KUKA KRL program: MyProgram_009().src

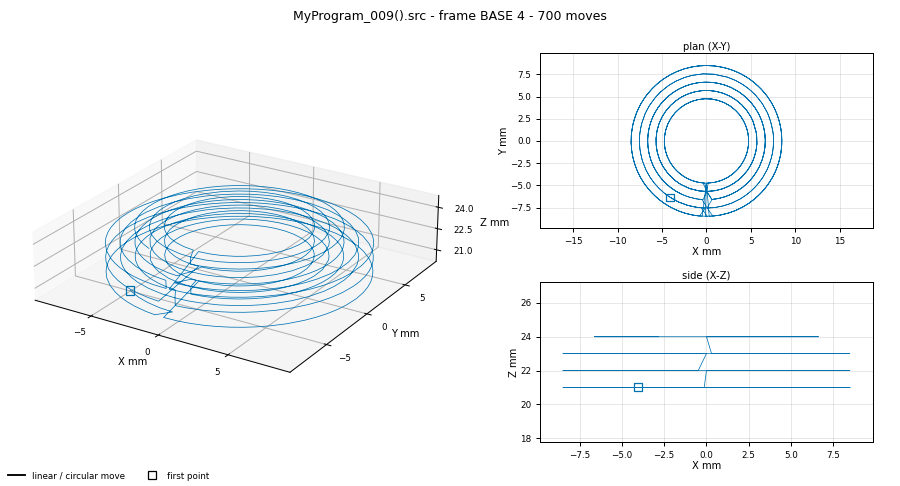
[picture p0: tool path of MyProgram_009().src in frame BASE 4, 700 of 700 moves have a stored position in this frame; points joined in program order, loops and branches not executed]
&ACCESS RVP
&REL 1
&PARAM TEMPLATE = C:\KRC\Roboter\Template\vorgabe
&PARAM EDITMASK = *
DEF MyProgram_009()
; ---- Setting reference (Base) ----
$BASE = BASE_DATA[4]

; --------------------------
; ---- Setting tool (TCP) ----
$TOOL = TOOL_DATA[3]
; --------------------------

$VEL.CP = VEL_APROX_PRINT
Startdeposition()
$VEL.CP = VEL_PRINT
LIN {X -4.0683,Y -6.363,Z 21,A -3.1712,B 0,C 0,E1 0.1598,E2 90.0712} C_DIS
LIN {X -3.0354,Y -6.9206,Z 21,A -3.1569,B 0,C 0,E1 0.1598,E2 90.0712} C_DIS
LIN {X -2.1485,Y -7.2456,Z 21,A -3.1382,B 0,C 0,E1 0.1598,E2 90.0713} C_DIS
LIN {X -1.0791,Y -7.4803,Z 21,A -3.109,B 0,C 0,E1 0.1598,E2 90.0713} C_DIS
LIN {X -0.0999,Y -7.555,Z 21,A -3.0763,B 0,C 0,E1 0.1598,E2 90.0715} C_DIS
Enddeposition()
LIN {X -0.0999,Y -7.555,Z 21,A -3.0763,B 0,C 0,E1 0.1598,E2 90.0715} C_DIS
Startdeposition()
$VEL.CP = VEL_PRINT
LIN {X -0.7948,Y -8.4503,Z 21,A -3.1394,B 0,C 0,E1 0.1598,E2 90.0708} C_DIS
LIN {X -1.524,Y -8.3542,Z 21,A -3.1626,B 0,C 0,E1 0.1598,E2 90.0713} C_DIS
LIN {X -2.5177,Y -8.1076,Z 21,A -3.1885,B 0,C 0,E1 0.1598,E2 90.0713} C_DIS
LIN {X -3.2872,Y -7.8268,Z 21,A -3.2048,B 0,C 0,E1 0.1598,E2 90.0713} C_DIS
LIN {X -4.0259,Y -7.4729,Z 21,A -3.2169,B 0,C 0,E1 0.1598,E2 90.0713} C_DIS
LIN {X -4.7269,Y -7.0495,Z 21,A -3.2247,B 0,C 0,E1 0.1598,E2 90.0712} C_DIS
LIN {X -5.5428,Y -6.4311,Z 21,A -3.2283,B 0,C 0,E1 0.1598,E2 90.071} C_DIS
LIN {X -6.3573,Y -5.629,Z 21,A -3.2241,B 0,C 0,E1 0.1598,E2 90.071} C_DIS
LIN {X -6.9724,Y -4.8392,Z 21,A -3.2134,B 0,C 0,E1 0.1598,E2 90.071} C_DIS
LIN {X -7.3967,Y -4.1598,Z 21,A -3.2003,B 0,C 0,E1 0.1598,E2 90.071} C_DIS
LIN {X -7.7565,Y -3.4443,Z 21,A -3.1833,B 0,C 0,E1 0.1598,E2 90.071} C_DIS
LIN {X -8.0474,Y -2.698,Z 21,A -3.1625,B 0,C 0,E1 0.1598,E2 90.071} C_DIS
LIN {X -8.2655,Y -1.9273,Z 21,A -3.138,B 0,C 0,E1 0.1598,E2 90.071} C_DIS
LIN {X -8.4101,Y -1.1396,Z 21,A -3.1101,B 0,C 0,E1 0.1598,E2 90.0711} C_DIS
LIN {X -8.4806,Y -0.3418,Z 21,A -3.079,B 0,C 0,E1 0.1598,E2 90.0711} C_DIS
LIN {X -8.4653,Y 0.6591,Z 21,A -3.036,B 0,C 0,E1 0.1598,E2 90.0709} C_DIS
LIN {X -8.2847,Y 1.8443,Z 21,A -2.9793,B 0,C 0,E1 0.1598,E2 90.0709} C_DIS
LIN {X -8.0734,Y 2.6138,Z 21,A -2.9395,B 0,C 0,E1 0.1598,E2 90.0713} C_DIS
LIN {X -7.7917,Y 3.3604,Z 21,A -2.8977,B 0,C 0,E1 0.1598,E2 90.0714} C_DIS
LIN {X -7.4414,Y 4.0773,Z 21,A -2.8546,B 0,C 0,E1 0.1598,E2 90.0715} C_DIS
LIN {X -7.0277,Y 4.7596,Z 21,A -2.8106,B 0,C 0,E1 0.1598,E2 90.0715} C_DIS
LIN {X -6.549,Y 5.3982,Z 21,A -2.7661,B 0,C 0,E1 0.1598,E2 90.0717} C_DIS
LIN {X -5.7701,Y 6.2287,Z 21,A -2.7022,B 0,C 0,E1 0.1598,E2 90.0717} C_DIS
LIN {X -4.9804,Y 6.8782,Z 21,A -2.6458,B 0,C 0,E1 0.1598,E2 90.0718} C_DIS
LIN {X -4.0916,Y 7.4385,Z 21,A -2.5895,B 0,C 0,E1 0.1598,E2 90.072} C_DIS
LIN {X -3.3359,Y 7.8065,Z 21,A -2.5461,B 0,C 0,E1 0.1598,E2 90.0721} C_DIS
LIN {X -2.5475,Y 8.0981,Z 21,A -2.5047,B 0,C 0,E1 0.1598,E2 90.0721} C_DIS
LIN {X -1.7342,Y 8.3101,Z 21,A -2.4658,B 0,C 0,E1 0.1598,E2 90.0723} C_DIS
LIN {X -0.9038,Y 8.44,Z 21,A -2.4296,B 0,C 0,E1 0.1598,E2 90.0723} C_DIS
LIN {X -0.0646,Y 8.4866,Z 21,A -2.3967,B 0,C 0,E1 0.1598,E2 90.0723} C_DIS
LIN {X 0.7752,Y 8.4513,Z 21,A -2.3671,B 0,C 0,E1 0.1598,E2 90.0724} C_DIS
LIN {X 1.6073,Y 8.3337,Z 21,A -2.3414,B 0,C 0,E1 0.1598,E2 90.0724} C_DIS
LIN {X 2.4237,Y 8.1342,Z 21,A -2.3196,B 0,C 0,E1 0.1598,E2 90.0724} C_DIS
LIN {X 3.2162,Y 7.8546,Z 21,A -2.3022,B 0,C 0,E1 0.1598,E2 90.0724} C_DIS
LIN {X 3.9771,Y 7.498,Z 21,A -2.2892,B 0,C 0,E1 0.1598,E2 90.0724} C_DIS
LIN {X 4.6991,Y 7.0679,Z 21,A -2.2807,B 0,C 0,E1 0.1598,E2 90.0724} C_DIS
LIN {X 5.3751,Y 6.5684,Z 21,A -2.2769,B 0,C 0,E1 0.1598,E2 90.0724} C_DIS
LIN {X 6.2322,Y 5.7664,Z 21,A -2.2791,B 0,C 0,E1 0.1598,E2 90.0722} C_DIS
LIN {X 6.8932,Y 4.9521,Z 21,A -2.2893,B 0,C 0,E1 0.1598,E2 90.0722} C_DIS
LIN {X 7.3483,Y 4.2471,Z 21,A -2.3025,B 0,C 0,E1 0.1598,E2 90.0722} C_DIS
LIN {X 7.7317,Y 3.5007,Z 21,A -2.3201,B 0,C 0,E1 0.1598,E2 90.0722} C_DIS
LIN {X 8.0395,Y 2.7201,Z 21,A -2.3419,B 0,C 0,E1 0.1598,E2 90.0721} C_DIS
LIN {X 8.2688,Y 1.913,Z 21,A -2.3677,B 0,C 0,E1 0.1598,E2 90.0721} C_DIS
LIN {X 8.4177,Y 1.0873,Z 21,A -2.3974,B 0,C 0,E1 0.1598,E2 90.072} C_DIS
LIN {X 8.4918,Y 0.0412,Z 21,A -2.4388,B 0,C 0,E1 0.1598,E2 90.0716} C_DIS
LIN {X 8.4127,Y -1.1163,Z 21,A -2.4909,B 0,C 0,E1 0.1598,E2 90.0715} C_DIS
LIN {X 8.2597,Y -1.9478,Z 21,A -2.5323,B 0,C 0,E1 0.1598,E2 90.0718} C_DIS
LIN {X 8.0253,Y -2.7601,Z 21,A -2.5755,B 0,C 0,E1 0.1598,E2 90.0718} C_DIS
LIN {X 7.7111,Y -3.5449,Z 21,A -2.6205,B 0,C 0,E1 0.1598,E2 90.0718} C_DIS
LIN {X 7.3199,Y -4.2944,Z 21,A -2.6668,B 0,C 0,E1 0.1598,E2 90.0718} C_DIS
LIN {X 6.6511,Y -5.2781,Z 21,A -2.733,B 0,C 0,E1 0.1598,E2 90.0715} C_DIS
LIN {X 5.9658,Y -6.0366,Z 21,A -2.7906,B 0,C 0,E1 0.1598,E2 90.0715} C_DIS
LIN {X 5.3564,Y -6.5819,Z 21,A -2.8363,B 0,C 0,E1 0.1598,E2 90.0716} C_DIS
LIN {X 4.6979,Y -7.0665,Z 21,A -2.8811,B 0,C 0,E1 0.1598,E2 90.0716} C_DIS
LIN {X 3.9958,Y -7.4856,Z 21,A -2.9247,B 0,C 0,E1 0.1598,E2 90.0716} C_DIS
LIN {X 3.2567,Y -7.8353,Z 21,A -2.9667,B 0,C 0,E1 0.1598,E2 90.0716} C_DIS
LIN {X 2.4875,Y -8.1124,Z 21,A -3.0067,B 0,C 0,E1 0.1598,E2 90.0716} C_DIS
LIN {X 1.6953,Y -8.3144,Z 21,A -3.0443,B 0,C 0,E1 0.1598,E2 90.0716} C_DIS
LIN {X 0.8873,Y -8.4397,Z 21,A -3.0793,B 0,C 0,E1 0.1598,E2 90.0715} C_DIS
LIN {X -0.1334,Y -8.4872,Z 21,A -3.1187,B 0,C 0,E1 0.1598,E2 90.0715} C_DIS
Enddeposition()
LIN {X 0.0005,Y -4.7572,Z 22,A -2.9405,B 0,C 0,E1 0.1598,E2 90.0604} C_DIS
Startdeposition()
$VEL.CP = VEL_PRINT
LIN {X 0.0005,Y -4.7572,Z 22,A -2.9462,B 0,C 0,E1 0.1598,E2 90.0661} C_DIS
LIN {X 0.9506,Y -4.6543,Z 22,A -2.9118,B 0,C 0,E1 0.1598,E2 90.071} C_DIS
LIN {X 1.6849,Y -4.4415,Z 22,A -2.8764,B 0,C 0,E1 0.1598,E2 90.0717} C_DIS
LIN {X 2.3764,Y -4.1152,Z 22,A -2.8372,B 0,C 0,E1 0.1598,E2 90.0717} C_DIS
LIN {X 3.0053,Y -3.68,Z 22,A -2.7955,B 0,C 0,E1 0.1598,E2 90.0717} C_DIS
LIN {X 3.5547,Y -3.1485,Z 22,A -2.7527,B 0,C 0,E1 0.1598,E2 90.0717} C_DIS
LIN {X 4.0149,Y -2.5382,Z 22,A -2.7099,B 0,C 0,E1 0.1598,E2 90.0717} C_DIS
LIN {X 4.37,Y -1.8612,Z 22,A -2.668,B 0,C 0,E1 0.1598,E2 90.0717} C_DIS
LIN {X 4.6111,Y -1.1359,Z 22,A -2.6283,B 0,C 0,E1 0.1598,E2 90.0717} C_DIS
LIN {X 4.734,Y -0.3815,Z 22,A -2.5917,B 0,C 0,E1 0.1598,E2 90.0718} C_DIS
LIN {X 4.7337,Y 0.3827,Z 22,A -2.5592,B 0,C 0,E1 0.1598,E2 90.0718} C_DIS
LIN {X 4.6108,Y 1.137,Z 22,A -2.5317,B 0,C 0,E1 0.1598,E2 90.0718} C_DIS
LIN {X 4.3693,Y 1.8622,Z 22,A -2.5099,B 0,C 0,E1 0.1598,E2 90.0719} C_DIS
LIN {X 4.0142,Y 2.5391,Z 22,A -2.4942,B 0,C 0,E1 0.1598,E2 90.0719} C_DIS
LIN {X 3.679,Y 3.0044,Z 22,A -2.487,B 0,C 0,E1 0.1598,E2 90.0721} C_DIS
LIN {X 3.1484,Y 3.5548,Z 22,A -2.4831,B 0,C 0,E1 0.1598,E2 90.0721} C_DIS
LIN {X 2.6975,Y 3.9089,Z 22,A -2.4848,B 0,C 0,E1 0.1598,E2 90.0721} C_DIS
LIN {X 2.0353,Y 4.2907,Z 22,A -2.4931,B 0,C 0,E1 0.1598,E2 90.0721} C_DIS
LIN {X 1.3208,Y 4.5621,Z 22,A -2.508,B 0,C 0,E1 0.1598,E2 90.0721} C_DIS
LIN {X 0.5721,Y 4.7168,Z 22,A -2.529,B 0,C 0,E1 0.1598,E2 90.0721} C_DIS
LIN {X -0.1919,Y 4.7486,Z 22,A -2.5559,B 0,C 0,E1 0.1598,E2 90.0721} C_DIS
LIN {X -0.9507,Y 4.6542,Z 22,A -2.5878,B 0,C 0,E1 0.1598,E2 90.0721} C_DIS
LIN {X -1.6845,Y 4.4401,Z 22,A -2.6239,B 0,C 0,E1 0.1598,E2 90.0721} C_DIS
LIN {X -2.3747,Y 4.112,Z 22,A -2.6632,B 0,C 0,E1 0.1598,E2 90.072} C_DIS
LIN {X -3.0046,Y 3.6789,Z 22,A -2.7047,B 0,C 0,E1 0.1598,E2 90.0719} C_DIS
LIN {X -3.5548,Y 3.1485,Z 22,A -2.7473,B 0,C 0,E1 0.1598,E2 90.0718} C_DIS
LIN {X -4.0153,Y 2.5384,Z 22,A -2.79,B 0,C 0,E1 0.1598,E2 90.0717} C_DIS
LIN {X -4.3701,Y 1.8612,Z 22,A -2.8316,B 0,C 0,E1 0.1598,E2 90.0716} C_DIS
LIN {X -4.6111,Y 1.1358,Z 22,A -2.8711,B 0,C 0,E1 0.1598,E2 90.0715} C_DIS
LIN {X -4.734,Y 0.3815,Z 22,A -2.9074,B 0,C 0,E1 0.1598,E2 90.0715} C_DIS
LIN {X -4.7346,Y -0.3828,Z 22,A -2.9397,B 0,C 0,E1 0.1598,E2 90.0713} C_DIS
LIN {X -4.611,Y -1.137,Z 22,A -2.967,B 0,C 0,E1 0.1598,E2 90.0713} C_DIS
LIN {X -4.3699,Y -1.8624,Z 22,A -2.9888,B 0,C 0,E1 0.1598,E2 90.0713} C_DIS
LIN {X -4.0147,Y -2.5393,Z 22,A -3.0044,B 0,C 0,E1 0.1598,E2 90.0713} C_DIS
LIN {X -3.5544,Y -3.1496,Z 22,A -3.0134,B 0,C 0,E1 0.1598,E2 90.0713} C_DIS
LIN {X -3.0038,Y -3.6798,Z 22,A -3.0156,B 0,C 0,E1 0.1598,E2 90.0713} C_DIS
LIN {X -2.3737,Y -4.1126,Z 22,A -3.0109,B 0,C 0,E1 0.1598,E2 90.0715} C_DIS
LIN {X -1.6836,Y -4.4408,Z 22,A -2.9995,B 0,C 0,E1 0.1598,E2 90.0715} C_DIS
LIN {X -0.9496,Y -4.6545,Z 22,A -2.9816,B 0,C 0,E1 0.1598,E2 90.0715} C_DIS
LIN {X -0.1908,Y -4.7488,Z 22,A -2.9578,B 0,C 0,E1 0.1598,E2 90.0716} C_DIS
LIN {X -0.1908,Y -4.7488,Z 22,A -2.9578,B 0,C 0,E1 0.1598,E2 90.0716} C_DIS
Enddeposition()
LIN {X 0.0239,Y -5.6874,Z 22,A -2.9887,B 0,C 0,E1 0.1598,E2 90.0704} C_DIS
Startdeposition()
$VEL.CP = VEL_PRINT
LIN {X -0.9077,Y -5.6101,Z 22,A -3.0207,B 0,C 0,E1 0.1598,E2 90.0715} C_DIS
LIN {X -1.8174,Y -5.3928,Z 22,A -3.0449,B 0,C 0,E1 0.1598,E2 90.0715} C_DIS
LIN {X -2.8689,Y -4.9093,Z 22,A -3.0629,B 0,C 0,E1 0.1598,E2 90.0714} C_DIS
LIN {X -3.4854,Y -4.493,Z 22,A -3.0679,B 0,C 0,E1 0.1598,E2 90.0714} C_DIS
LIN {X -4.2717,Y -3.7584,Z 22,A -3.0655,B 0,C 0,E1 0.1598,E2 90.0712} C_DIS
LIN {X -4.9659,Y -2.7683,Z 22,A -3.0489,B 0,C 0,E1 0.1598,E2 90.071} C_DIS
LIN {X -5.3072,Y -2.0335,Z 22,A -3.0306,B 0,C 0,E1 0.1598,E2 90.0712} C_DIS
LIN {X -5.5422,Y -1.2582,Z 22,A -3.0065,B 0,C 0,E1 0.1598,E2 90.0712} C_DIS
LIN {X -5.6647,Y -0.4576,Z 22,A -2.9772,B 0,C 0,E1 0.1598,E2 90.0712} C_DIS
LIN {X -5.671,Y 0.3523,Z 22,A -2.9432,B 0,C 0,E1 0.1598,E2 90.0713} C_DIS
LIN {X -5.5643,Y 1.1551,Z 22,A -2.9054,B 0,C 0,E1 0.1598,E2 90.0713} C_DIS
LIN {X -5.3438,Y 1.9345,Z 22,A -2.8644,B 0,C 0,E1 0.1598,E2 90.0714} C_DIS
LIN {X -5.0149,Y 2.6749,Z 22,A -2.8211,B 0,C 0,E1 0.1598,E2 90.0715} C_DIS
LIN {X -4.5827,Y 3.3599,Z 22,A -2.7763,B 0,C 0,E1 0.1598,E2 90.0716} C_DIS
LIN {X -4.0594,Y 3.9784,Z 22,A -2.7309,B 0,C 0,E1 0.1598,E2 90.0717} C_DIS
LIN {X -3.4528,Y 4.5155,Z 22,A -2.6859,B 0,C 0,E1 0.1598,E2 90.0718} C_DIS
LIN {X -2.7758,Y 4.9605,Z 22,A -2.6422,B 0,C 0,E1 0.1598,E2 90.072} C_DIS
LIN {X -2.0422,Y 5.3045,Z 22,A -2.6007,B 0,C 0,E1 0.1598,E2 90.072} C_DIS
LIN {X -1.2671,Y 5.54,Z 22,A -2.5622,B 0,C 0,E1 0.1598,E2 90.0721} C_DIS
LIN {X -0.4666,Y 5.6638,Z 22,A -2.5274,B 0,C 0,E1 0.1598,E2 90.0721} C_DIS
LIN {X 0.3433,Y 5.6719,Z 22,A -2.4972,B 0,C 0,E1 0.1598,E2 90.0722} C_DIS
LIN {X 1.1461,Y 5.5657,Z 22,A -2.4721,B 0,C 0,E1 0.1598,E2 90.0722} C_DIS
LIN {X 1.9259,Y 5.3468,Z 22,A -2.4526,B 0,C 0,E1 0.1598,E2 90.0722} C_DIS
LIN {X 2.6663,Y 5.0183,Z 22,A -2.4392,B 0,C 0,E1 0.1598,E2 90.0722} C_DIS
LIN {X 3.3528,Y 4.5884,Z 22,A -2.432,B 0,C 0,E1 0.1598,E2 90.0722} C_DIS
LIN {X 3.9712,Y 4.0652,Z 22,A -2.4314,B 0,C 0,E1 0.1598,E2 90.0722} C_DIS
LIN {X 4.5093,Y 3.4597,Z 22,A -2.4372,B 0,C 0,E1 0.1598,E2 90.0722} C_DIS
LIN {X 4.9567,Y 2.7841,Z 22,A -2.4493,B 0,C 0,E1 0.1598,E2 90.072} C_DIS
LIN {X 5.2296,Y 2.2406,Z 22,A -2.4624,B 0,C 0,E1 0.1598,E2 90.0721} C_DIS
LIN {X 5.6357,Y 0.7895,Z 22,A -2.5081,B 0,C 0,E1 0.1598,E2 90.0711} C_DIS
LIN {X 5.6765,Y -0.309,Z 22,A -2.5537,B 0,C 0,E1 0.1598,E2 90.0714} C_DIS
LIN {X 5.5814,Y -1.0665,Z 22,A -2.5897,B 0,C 0,E1 0.1598,E2 90.0718} C_DIS
LIN {X 5.391,Y -1.8058,Z 22,A -2.6282,B 0,C 0,E1 0.1598,E2 90.0718} C_DIS
LIN {X 5.099,Y -2.5114,Z 22,A -2.669,B 0,C 0,E1 0.1598,E2 90.0718} C_DIS
LIN {X 4.7183,Y -3.173,Z 22,A -2.7111,B 0,C 0,E1 0.1598,E2 90.0718} C_DIS
LIN {X 4.2493,Y -3.7757,Z 22,A -2.754,B 0,C 0,E1 0.1598,E2 90.0718} C_DIS
LIN {X 3.7051,Y -4.3113,Z 22,A -2.7968,B 0,C 0,E1 0.1598,E2 90.0718} C_DIS
LIN {X 3.0932,Y -4.7678,Z 22,A -2.8387,B 0,C 0,E1 0.1598,E2 90.0717} C_DIS
LIN {X 2.426,Y -5.1388,Z 22,A -2.8789,B 0,C 0,E1 0.1598,E2 90.0717} C_DIS
LIN {X 1.7156,Y -5.4181,Z 22,A -2.9169,B 0,C 0,E1 0.1598,E2 90.0717} C_DIS
LIN {X 0.9745,Y -5.6021,Z 22,A -2.9519,B 0,C 0,E1 0.1598,E2 90.0717} C_DIS
LIN {X 0.0239,Y -5.6874,Z 22,A -2.9904,B 0,C 0,E1 0.1598,E2 90.0716} C_DIS
Enddeposition()
LIN {X 0.0239,Y -5.6874,Z 22,A -2.9904,B 0,C 0,E1 0.1598,E2 90.0716} C_DIS
Startdeposition()
$VEL.CP = VEL_PRINT
LIN {X 0.6181,Y -6.5909,Z 22,A -3.0065,B 0,C 0,E1 0.1598,E2 90.071} C_DIS
LIN {X 1.3584,Y -6.477,Z 22,A -2.9751,B 0,C 0,E1 0.1598,E2 90.0716} C_DIS
LIN {X 2.082,Y -6.284,Z 22,A -2.9404,B 0,C 0,E1 0.1598,E2 90.0716} C_DIS
LIN {X 2.7786,Y -6.0085,Z 22,A -2.9031,B 0,C 0,E1 0.1598,E2 90.0716} C_DIS
LIN {X 3.4393,Y -5.656,Z 22,A -2.8638,B 0,C 0,E1 0.1598,E2 90.0716} C_DIS
LIN {X 4.0554,Y -5.2301,Z 22,A -2.8231,B 0,C 0,E1 0.1598,E2 90.0717} C_DIS
LIN {X 4.621,Y -4.7391,Z 22,A -2.7814,B 0,C 0,E1 0.1598,E2 90.0717} C_DIS
LIN {X 5.1275,Y -4.1872,Z 22,A -2.7393,B 0,C 0,E1 0.1598,E2 90.0717} C_DIS
LIN {X 5.5674,Y -3.581,Z 22,A -2.6974,B 0,C 0,E1 0.1598,E2 90.0717} C_DIS
LIN {X 5.9348,Y -2.9284,Z 22,A -2.6561,B 0,C 0,E1 0.1598,E2 90.0718} C_DIS
LIN {X 6.2272,Y -2.239,Z 22,A -2.616,B 0,C 0,E1 0.1598,E2 90.0718} C_DIS
LIN {X 6.4419,Y -1.5216,Z 22,A -2.5776,B 0,C 0,E1 0.1598,E2 90.0718} C_DIS
LIN {X 6.5734,Y -0.7842,Z 22,A -2.5414,B 0,C 0,E1 0.1598,E2 90.0718} C_DIS
LIN {X 6.6187,Y -0.0366,Z 22,A -2.5079,B 0,C 0,E1 0.1598,E2 90.0719} C_DIS
LIN {X 6.5802,Y 0.7112,Z 22,A -2.4775,B 0,C 0,E1 0.1598,E2 90.0719} C_DIS
LIN {X 6.4572,Y 1.45,Z 22,A -2.4506,B 0,C 0,E1 0.1598,E2 90.0719} C_DIS
LIN {X 6.2523,Y 2.1702,Z 22,A -2.4276,B 0,C 0,E1 0.1598,E2 90.072} C_DIS
LIN {X 5.9671,Y 2.8627,Z 22,A -2.4087,B 0,C 0,E1 0.1598,E2 90.072} C_DIS
LIN {X 5.6048,Y 3.5181,Z 22,A -2.3942,B 0,C 0,E1 0.1598,E2 90.0721} C_DIS
LIN {X 5.1721,Y 4.1292,Z 22,A -2.3843,B 0,C 0,E1 0.1598,E2 90.0721} C_DIS
LIN {X 4.6732,Y 4.6877,Z 22,A -2.379,B 0,C 0,E1 0.1598,E2 90.0722} C_DIS
LIN {X 4.1131,Y 5.185,Z 22,A -2.3786,B 0,C 0,E1 0.1598,E2 90.0722} C_DIS
LIN {X 3.5008,Y 5.6164,Z 22,A -2.3829,B 0,C 0,E1 0.1598,E2 90.0722} C_DIS
LIN {X 2.8448,Y 5.9776,Z 22,A -2.3919,B 0,C 0,E1 0.1598,E2 90.0722} C_DIS
LIN {X 2.1507,Y 6.2591,Z 22,A -2.4056,B 0,C 0,E1 0.1598,E2 90.0723} C_DIS
LIN {X 1.4298,Y 6.4619,Z 22,A -2.4236,B 0,C 0,E1 0.1598,E2 90.0723} C_DIS
LIN {X 0.6907,Y 6.5828,Z 22,A -2.4458,B 0,C 0,E1 0.1598,E2 90.0723} C_DIS
LIN {X -0.0573,Y 6.6184,Z 22,A -2.4719,B 0,C 0,E1 0.1598,E2 90.0723} C_DIS
LIN {X -0.8046,Y 6.5698,Z 22,A -2.5015,B 0,C 0,E1 0.1598,E2 90.0723} C_DIS
LIN {X -1.5414,Y 6.4358,Z 22,A -2.5344,B 0,C 0,E1 0.1598,E2 90.0722} C_DIS
LIN {X -2.2586,Y 6.2203,Z 22,A -2.5699,B 0,C 0,E1 0.1598,E2 90.0722} C_DIS
LIN {X -2.9478,Y 5.9273,Z 22,A -2.6077,B 0,C 0,E1 0.1598,E2 90.0721} C_DIS
LIN {X -3.5981,Y 5.556,Z 22,A -2.6473,B 0,C 0,E1 0.1598,E2 90.072} C_DIS
LIN {X -4.203,Y 5.1142,Z 22,A -2.6882,B 0,C 0,E1 0.1598,E2 90.0719} C_DIS
LIN {X -4.7547,Y 4.6076,Z 22,A -2.7299,B 0,C 0,E1 0.1598,E2 90.0719} C_DIS
LIN {X -5.2454,Y 4.0418,Z 22,A -2.7719,B 0,C 0,E1 0.1598,E2 90.0717} C_DIS
LIN {X -5.6675,Y 3.423,Z 22,A -2.8135,B 0,C 0,E1 0.1598,E2 90.0717} C_DIS
LIN {X -6.0163,Y 2.7603,Z 22,A -2.8542,B 0,C 0,E1 0.1598,E2 90.0715} C_DIS
LIN {X -6.2888,Y 2.0627,Z 22,A -2.8937,B 0,C 0,E1 0.1598,E2 90.0715} C_DIS
LIN {X -6.4824,Y 1.3391,Z 22,A -2.9313,B 0,C 0,E1 0.1598,E2 90.0714} C_DIS
LIN {X -6.5915,Y 0.5982,Z 22,A -2.9666,B 0,C 0,E1 0.1598,E2 90.0714} C_DIS
LIN {X -6.6178,Y -0.1502,Z 22,A -2.9991,B 0,C 0,E1 0.1598,E2 90.0713} C_DIS
LIN {X -6.5564,Y -0.8967,Z 22,A -3.0283,B 0,C 0,E1 0.1598,E2 90.0713} C_DIS
LIN {X -6.4138,Y -1.6318,Z 22,A -3.0541,B 0,C 0,E1 0.1598,E2 90.0713} C_DIS
LIN {X -6.1902,Y -2.3465,Z 22,A -3.0761,B 0,C 0,E1 0.1598,E2 90.0713} C_DIS
LIN {X -5.8854,Y -3.0308,Z 22,A -3.0938,B 0,C 0,E1 0.1598,E2 90.0713} C_DIS
LIN {X -5.5049,Y -3.6762,Z 22,A -3.1072,B 0,C 0,E1 0.1598,E2 90.0713} C_DIS
LIN {X -5.0542,Y -4.2744,Z 22,A -3.1159,B 0,C 0,E1 0.1598,E2 90.0713} C_DIS
LIN {X -4.5381,Y -4.8171,Z 22,A -3.12,B 0,C 0,E1 0.1598,E2 90.0713} C_DIS
LIN {X -3.9654,Y -5.2996,Z 22,A -3.1194,B 0,C 0,E1 0.1598,E2 90.0713} C_DIS
LIN {X -3.3417,Y -5.7143,Z 22,A -3.1141,B 0,C 0,E1 0.1598,E2 90.0713} C_DIS
LIN {X -2.6743,Y -6.0543,Z 22,A -3.104,B 0,C 0,E1 0.1598,E2 90.0713} C_DIS
LIN {X -1.9731,Y -6.3174,Z 22,A -3.0895,B 0,C 0,E1 0.1598,E2 90.0714} C_DIS
LIN {X -1.2466,Y -6.4991,Z 22,A -3.0705,B 0,C 0,E1 0.1598,E2 90.0714} C_DIS
LIN {X -0.5044,Y -6.5992,Z 22,A -3.0476,B 0,C 0,E1 0.1598,E2 90.0715} C_DIS
LIN {X -0.5044,Y -6.5992,Z 22,A -3.0476,B 0,C 0,E1 0.1598,E2 90.0715} C_DIS
Enddeposition()
LIN {X 0.094,Y -7.5561,Z 22,A -3.0652,B 0,C 0,E1 0.1598,E2 90.0703} C_DIS
Startdeposition()
$VEL.CP = VEL_PRINT
LIN {X -0.9287,Y -7.4999,Z 22,A -3.1014,B 0,C 0,E1 0.1598,E2 90.0714} C_DIS
LIN {X -2.0681,Y -7.2643,Z 22,A -3.1332,B 0,C 0,E1 0.1598,E2 90.0714} C_DIS
LIN {X -3.1208,Y -6.8842,Z 22,A -3.1557,B 0,C 0,E1 0.1598,E2 90.0713} C_DIS
LIN {X -3.8898,Y -6.4791,Z 22,A -3.1667,B 0,C 0,E1 0.1598,E2 90.0713} C_DIS
LIN {X -4.7183,Y -5.8987,Z 22,A -3.1725,B 0,C 0,E1 0.1598,E2 90.0712} C_DIS
LIN {X -5.3217,Y -5.3594,Z 22,A -3.1718,B 0,C 0,E1 0.1598,E2 90.0712} C_DIS
LIN {X -5.8648,Y -4.7594,Z 22,A -3.1664,B 0,C 0,E1 0.1598,E2 90.0712} C_DIS
LIN {X -6.3392,Y -4.1039,Z 22,A -3.1561,B 0,C 0,E1 0.1598,E2 90.0712} C_DIS
LIN {X -6.8355,Y -3.2224,Z 22,A -3.1368,B 0,C 0,E1 0.1598,E2 90.0709} C_DIS
LIN {X -7.2583,Y -2.0894,Z 22,A -3.1043,B 0,C 0,E1 0.1598,E2 90.0707} C_DIS
LIN {X -7.4986,Y -0.9403,Z 22,A -3.0647,B 0,C 0,E1 0.1598,E2 90.0708} C_DIS
LIN {X -7.5583,Y -0.0227,Z 22,A -3.0283,B 0,C 0,E1 0.1598,E2 90.071} C_DIS
LIN {X -7.4851,Y 1.0498,Z 22,A -2.9803,B 0,C 0,E1 0.1598,E2 90.071} C_DIS
LIN {X -7.2636,Y 2.0716,Z 22,A -2.9291,B 0,C 0,E1 0.1598,E2 90.0712} C_DIS
LIN {X -6.8715,Y 3.1482,Z 22,A -2.8692,B 0,C 0,E1 0.1598,E2 90.0712} C_DIS
LIN {X -6.4236,Y 3.9796,Z 22,A -2.8179,B 0,C 0,E1 0.1598,E2 90.0715} C_DIS
LIN {X -5.7272,Y 4.9293,Z 22,A -2.752,B 0,C 0,E1 0.1598,E2 90.0715} C_DIS
LIN {X -5.1344,Y 5.5449,Z 22,A -2.7044,B 0,C 0,E1 0.1598,E2 90.0717} C_DIS
LIN {X -4.2688,Y 6.2352,Z 22,A -2.6434,B 0,C 0,E1 0.1598,E2 90.0718} C_DIS
LIN {X -3.4769,Y 6.7108,Z 22,A -2.5942,B 0,C 0,E1 0.1598,E2 90.072} C_DIS
LIN {X -2.4258,Y 7.1536,Z 22,A -2.5368,B 0,C 0,E1 0.1598,E2 90.072} C_DIS
LIN {X -1.7381,Y 7.356,Z 22,A -2.5029,B 0,C 0,E1 0.1598,E2 90.0722} C_DIS
LIN {X -0.3701,Y 7.5491,Z 22,A -2.4443,B 0,C 0,E1 0.1598,E2 90.0722} C_DIS
LIN {X 0.834,Y 7.5107,Z 22,A -2.4014,B 0,C 0,E1 0.1598,E2 90.0724} C_DIS
LIN {X 2.4072,Y 7.1599,Z 22,A -2.3581,B 0,C 0,E1 0.1598,E2 90.0724} C_DIS
LIN {X 3.1208,Y 6.8791,Z 22,A -2.3437,B 0,C 0,E1 0.1598,E2 90.0724} C_DIS
LIN {X 3.8016,Y 6.5265,Z 22,A -2.3335,B 0,C 0,E1 0.1598,E2 90.0724} C_DIS
LIN {X 4.4438,Y 6.1075,Z 22,A -2.3275,B 0,C 0,E1 0.1598,E2 90.0724} C_DIS
LIN {X 5.0402,Y 5.6256,Z 22,A -2.3259,B 0,C 0,E1 0.1598,E2 90.0724} C_DIS
LIN {X 5.5852,Y 5.0861,Z 22,A -2.3287,B 0,C 0,E1 0.1598,E2 90.0723} C_DIS
LIN {X 6.3384,Y 4.1174,Z 22,A -2.3417,B 0,C 0,E1 0.1598,E2 90.0719} C_DIS
LIN {X 6.8151,Y 3.261,Z 22,A -2.3606,B 0,C 0,E1 0.1598,E2 90.0719} C_DIS
LIN {X 7.1191,Y 2.5351,Z 22,A -2.3803,B 0,C 0,E1 0.1598,E2 90.072} C_DIS
LIN {X 7.4889,Y 1.0245,Z 22,A -2.4299,B 0,C 0,E1 0.1598,E2 90.071} C_DIS
LIN {X 7.556,Y 0.1285,Z 22,A -2.4664,B 0,C 0,E1 0.1598,E2 90.0718} C_DIS
LIN {X 7.49,Y -0.9739,Z 22,A -2.5155,B 0,C 0,E1 0.1598,E2 90.0715} C_DIS
LIN {X 7.305,Y -1.9342,Z 22,A -2.5633,B 0,C 0,E1 0.1598,E2 90.0715} C_DIS
LIN {X 6.9014,Y -3.0686,Z 22,A -2.6262,B 0,C 0,E1 0.1598,E2 90.0713} C_DIS
LIN {X 6.3381,Y -4.118,Z 22,A -2.6917,B 0,C 0,E1 0.1598,E2 90.0714} C_DIS
LIN {X 5.6644,Y -4.9964,Z 22,A -2.7539,B 0,C 0,E1 0.1598,E2 90.0714} C_DIS
LIN {X 5.0977,Y -5.5737,Z 22,A -2.7995,B 0,C 0,E1 0.1598,E2 90.0717} C_DIS
LIN {X 4.472,Y -6.0863,Z 22,A -2.8443,B 0,C 0,E1 0.1598,E2 90.0717} C_DIS
LIN {X 3.7954,Y -6.5296,Z 22,A -2.888,B 0,C 0,E1 0.1598,E2 90.0717} C_DIS
LIN {X 2.8911,Y -6.982,Z 22,A -2.9404,B 0,C 0,E1 0.1598,E2 90.0716} C_DIS
LIN {X 1.7204,Y -7.3546,Z 22,A -2.9992,B 0,C 0,E1 0.1598,E2 90.0716} C_DIS
LIN {X 0.9762,Y -7.4946,Z 22,A -3.0325,B 0,C 0,E1 0.1598,E2 90.0716} C_DIS
LIN {X 0.094,Y -7.5561,Z 22,A -3.0675,B 0,C 0,E1 0.1598,E2 90.0715} C_DIS
Enddeposition()
LIN {X 0.094,Y -7.5561,Z 22,A -3.0675,B 0,C 0,E1 0.1598,E2 90.0715} C_DIS
Startdeposition()
$VEL.CP = VEL_PRINT
LIN {X 0.7148,Y -8.4578,Z 22,A -3.0826,B 0,C 0,E1 0.1598,E2 90.0709} C_DIS
LIN {X 1.4889,Y -8.36,Z 22,A -3.0506,B 0,C 0,E1 0.1598,E2 90.0715} C_DIS
LIN {X 2.4939,Y -8.1145,Z 22,A -3.0034,B 0,C 0,E1 0.1598,E2 90.0715} C_DIS
LIN {X 3.2722,Y -7.8328,Z 22,A -2.9629,B 0,C 0,E1 0.1598,E2 90.0715} C_DIS
LIN {X 4.0192,Y -7.4765,Z 22,A -2.9203,B 0,C 0,E1 0.1598,E2 90.0716} C_DIS
LIN {X 4.7278,Y -7.0489,Z 22,A -2.8761,B 0,C 0,E1 0.1598,E2 90.0716} C_DIS
LIN {X 5.3917,Y -6.5546,Z 22,A -2.8307,B 0,C 0,E1 0.1598,E2 90.0716} C_DIS
LIN {X 6.2364,Y -5.762,Z 22,A -2.7658,B 0,C 0,E1 0.1598,E2 90.0716} C_DIS
LIN {X 6.8899,Y -4.9637,Z 22,A -2.7078,B 0,C 0,E1 0.1598,E2 90.0716} C_DIS
LIN {X 7.4501,Y -4.0702,Z 22,A -2.6491,B 0,C 0,E1 0.1598,E2 90.0716} C_DIS
LIN {X 7.8174,Y -3.3107,Z 22,A -2.6034,B 0,C 0,E1 0.1598,E2 90.0718} C_DIS
LIN {X 8.1074,Y -2.5184,Z 22,A -2.559,B 0,C 0,E1 0.1598,E2 90.0718} C_DIS
LIN {X 8.3592,Y -1.4943,Z 22,A -2.5058,B 0,C 0,E1 0.1598,E2 90.0716} C_DIS
LIN {X 8.4809,Y -0.3252,Z 22,A -2.4514,B 0,C 0,E1 0.1598,E2 90.0716} C_DIS
LIN {X 8.4728,Y 0.4965,Z 22,A -2.4171,B 0,C 0,E1 0.1598,E2 90.0719} C_DIS
LIN {X 8.3859,Y 1.3137,Z 22,A -2.3856,B 0,C 0,E1 0.1598,E2 90.072} C_DIS
LIN {X 8.2205,Y 2.1187,Z 22,A -2.3574,B 0,C 0,E1 0.1598,E2 90.072} C_DIS
LIN {X 7.9769,Y 2.9037,Z 22,A -2.333,B 0,C 0,E1 0.1598,E2 90.072} C_DIS
LIN {X 7.6584,Y 3.6612,Z 22,A -2.3126,B 0,C 0,E1 0.1598,E2 90.0721} C_DIS
LIN {X 7.2682,Y 4.3845,Z 22,A -2.2962,B 0,C 0,E1 0.1598,E2 90.0721} C_DIS
LIN {X 6.8091,Y 5.066,Z 22,A -2.2842,B 0,C 0,E1 0.1598,E2 90.0722} C_DIS
LIN {X 6.1495,Y 5.8536,Z 22,A -2.275,B 0,C 0,E1 0.1598,E2 90.0722} C_DIS
LIN {X 5.2802,Y 6.6453,Z 22,A -2.2735,B 0,C 0,E1 0.1598,E2 90.0722} C_DIS
LIN {X 4.589,Y 7.1393,Z 22,A -2.2783,B 0,C 0,E1 0.1598,E2 90.0724} C_DIS
LIN {X 3.8525,Y 7.5624,Z 22,A -2.2876,B 0,C 0,E1 0.1598,E2 90.0724} C_DIS
LIN {X 3.0772,Y 7.9096,Z 22,A -2.3015,B 0,C 0,E1 0.1598,E2 90.0724} C_DIS
LIN {X 2.2712,Y 8.178,Z 22,A -2.32,B 0,C 0,E1 0.1598,E2 90.0724} C_DIS
LIN {X 1.0543,Y 8.4253,Z 22,A -2.3545,B 0,C 0,E1 0.1598,E2 90.0724} C_DIS
LIN {X -0.0055,Y 8.4875,Z 22,A -2.391,B 0,C 0,E1 0.1598,E2 90.0724} C_DIS
LIN {X -0.8537,Y 8.4448,Z 22,A -2.4241,B 0,C 0,E1 0.1598,E2 90.0724} C_DIS
LIN {X -1.6935,Y 8.3181,Z 22,A -2.4605,B 0,C 0,E1 0.1598,E2 90.0723} C_DIS
LIN {X -2.5163,Y 8.1076,Z 22,A -2.4997,B 0,C 0,E1 0.1598,E2 90.0723} C_DIS
LIN {X -3.3138,Y 7.8155,Z 22,A -2.5415,B 0,C 0,E1 0.1598,E2 90.0721} C_DIS
LIN {X -4.0783,Y 7.4455,Z 22,A -2.5853,B 0,C 0,E1 0.1598,E2 90.0721} C_DIS
LIN {X -4.8008,Y 6.9993,Z 22,A -2.6308,B 0,C 0,E1 0.1598,E2 90.072} C_DIS
LIN {X -5.4752,Y 6.4831,Z 22,A -2.6774,B 0,C 0,E1 0.1598,E2 90.0719} C_DIS
LIN {X -6.0957,Y 5.9034,Z 22,A -2.7247,B 0,C 0,E1 0.1598,E2 90.0718} C_DIS
LIN {X -6.6555,Y 5.2648,Z 22,A -2.7722,B 0,C 0,E1 0.1598,E2 90.0717} C_DIS
LIN {X -7.1494,Y 4.5739,Z 22,A -2.8195,B 0,C 0,E1 0.1598,E2 90.0716} C_DIS
LIN {X -7.57,Y 3.8362,Z 22,A -2.866,B 0,C 0,E1 0.1598,E2 90.0715} C_DIS
LIN {X -7.9157,Y 3.0604,Z 22,A -2.9114,B 0,C 0,E1 0.1598,E2 90.0714} C_DIS
LIN {X -8.2741,Y 1.9114,Z 22,A -2.9727,B 0,C 0,E1 0.1598,E2 90.071} C_DIS
LIN {X -8.4497,Y 0.8392,Z 22,A -3.0244,B 0,C 0,E1 0.1598,E2 90.071} C_DIS
LIN {X -8.4867,Y -0.1724,Z 22,A -3.0685,B 0,C 0,E1 0.1598,E2 90.071} C_DIS
LIN {X -8.43,Y -0.9801,Z 22,A -3.1006,B 0,C 0,E1 0.1598,E2 90.071} C_DIS
LIN {X -8.2993,Y -1.7793,Z 22,A -3.1295,B 0,C 0,E1 0.1598,E2 90.071} C_DIS
LIN {X -8.0929,Y -2.5623,Z 22,A -3.1549,B 0,C 0,E1 0.1598,E2 90.071} C_DIS
LIN {X -7.8113,Y -3.3217,Z 22,A -3.1766,B 0,C 0,E1 0.1598,E2 90.071} C_DIS
LIN {X -7.4601,Y -4.0513,Z 22,A -3.1946,B 0,C 0,E1 0.1598,E2 90.071} C_DIS
LIN {X -7.0388,Y -4.7429,Z 22,A -3.2083,B 0,C 0,E1 0.1598,E2 90.071} C_DIS
LIN {X -6.5543,Y -5.3918,Z 22,A -3.218,B 0,C 0,E1 0.1598,E2 90.071} C_DIS
LIN {X -5.7708,Y -6.2281,Z 22,A -3.2244,B 0,C 0,E1 0.1598,E2 90.071} C_DIS
LIN {X -4.9885,Y -6.8657,Z 22,A -3.2229,B 0,C 0,E1 0.1598,E2 90.071} C_DIS
LIN {X -4.3132,Y -7.3081,Z 22,A -3.2169,B 0,C 0,E1 0.1598,E2 90.0712} C_DIS
LIN {X -3.599,Y -7.6845,Z 22,A -3.2067,B 0,C 0,E1 0.1598,E2 90.0712} C_DIS
LIN {X -2.8525,Y -7.9916,Z 22,A -3.1924,B 0,C 0,E1 0.1598,E2 90.0712} C_DIS
LIN {X -2.0802,Y -8.2265,Z 22,A -3.174,B 0,C 0,E1 0.1598,E2 90.0713} C_DIS
LIN {X -1.2892,Y -8.3874,Z 22,A -3.1519,B 0,C 0,E1 0.1598,E2 90.0713} C_DIS
LIN {X -0.4865,Y -8.4731,Z 22,A -3.1261,B 0,C 0,E1 0.1598,E2 90.0714} C_DIS
LIN {X -0.4865,Y -8.4731,Z 22,A -3.1261,B 0,C 0,E1 0.1598,E2 90.0714} C_DIS
Enddeposition()
LIN {X 0.0005,Y -4.7523,Z 23,A -2.9353,B 0,C 0,E1 0.1598,E2 90.0603} C_DIS
Startdeposition()
$VEL.CP = VEL_PRINT
LIN {X 0.0005,Y -4.7523,Z 23,A -2.941,B 0,C 0,E1 0.1598,E2 90.0661} C_DIS
LIN {X -0.7613,Y -4.6869,Z 23,A -2.9711,B 0,C 0,E1 0.1598,E2 90.0709} C_DIS
LIN {X -1.3209,Y -4.5621,Z 23,A -2.987,B 0,C 0,E1 0.1598,E2 90.0715} C_DIS
LIN {X -2.0354,Y -4.2906,Z 23,A -3.0017,B 0,C 0,E1 0.1598,E2 90.0715} C_DIS
LIN {X -2.6978,Y -3.9092,Z 23,A -3.0098,B 0,C 0,E1 0.1598,E2 90.0715} C_DIS
LIN {X -3.2894,Y -3.4254,Z 23,A -3.011,B 0,C 0,E1 0.1598,E2 90.0715} C_DIS
LIN {X -3.6791,Y -3.0043,Z 23,A -3.0076,B 0,C 0,E1 0.1598,E2 90.0715} C_DIS
LIN {X -4.112,Y -2.3746,Z 23,A -2.9967,B 0,C 0,E1 0.1598,E2 90.0714} C_DIS
LIN {X -4.4398,Y -1.6844,Z 23,A -2.9795,B 0,C 0,E1 0.1598,E2 90.0714} C_DIS
LIN {X -4.6537,Y -0.9507,Z 23,A -2.9564,B 0,C 0,E1 0.1598,E2 90.0714} C_DIS
LIN {X -4.7408,Y -0.2874,Z 23,A -2.9316,B 0,C 0,E1 0.1598,E2 90.0714} C_DIS
LIN {X -4.7339,Y 0.3814,Z 23,A -2.903,B 0,C 0,E1 0.1598,E2 90.0714} C_DIS
LIN {X -4.6111,Y 1.1358,Z 23,A -2.8666,B 0,C 0,E1 0.1598,E2 90.0714} C_DIS
LIN {X -4.3701,Y 1.8612,Z 23,A -2.8271,B 0,C 0,E1 0.1598,E2 90.0715} C_DIS
LIN {X -4.0154,Y 2.5384,Z 23,A -2.7855,B 0,C 0,E1 0.1598,E2 90.0716} C_DIS
LIN {X -3.5548,Y 3.1485,Z 23,A -2.7428,B 0,C 0,E1 0.1598,E2 90.0717} C_DIS
LIN {X -3.0046,Y 3.6789,Z 23,A -2.7002,B 0,C 0,E1 0.1598,E2 90.0718} C_DIS
LIN {X -2.3747,Y 4.1119,Z 23,A -2.6587,B 0,C 0,E1 0.1598,E2 90.0719} C_DIS
LIN {X -1.6846,Y 4.4402,Z 23,A -2.6194,B 0,C 0,E1 0.1598,E2 90.072} C_DIS
LIN {X -0.9507,Y 4.6541,Z 23,A -2.5834,B 0,C 0,E1 0.1598,E2 90.0721} C_DIS
LIN {X -0.192,Y 4.7487,Z 23,A -2.5514,B 0,C 0,E1 0.1598,E2 90.0721} C_DIS
LIN {X 0.572,Y 4.7168,Z 23,A -2.5246,B 0,C 0,E1 0.1598,E2 90.0722} C_DIS
LIN {X 1.3208,Y 4.5621,Z 23,A -2.5035,B 0,C 0,E1 0.1598,E2 90.0722} C_DIS
LIN {X 2.0353,Y 4.2907,Z 23,A -2.4886,B 0,C 0,E1 0.1598,E2 90.0722} C_DIS
LIN {X 2.6974,Y 3.909,Z 23,A -2.4804,B 0,C 0,E1 0.1598,E2 90.0722} C_DIS
LIN {X 3.2893,Y 3.4255,Z 23,A -2.479,B 0,C 0,E1 0.1598,E2 90.0722} C_DIS
LIN {X 3.679,Y 3.0044,Z 23,A -2.4825,B 0,C 0,E1 0.1598,E2 90.0722} C_DIS
LIN {X 4.1119,Y 2.3747,Z 23,A -2.4932,B 0,C 0,E1 0.1598,E2 90.072} C_DIS
LIN {X 4.4397,Y 1.6844,Z 23,A -2.5104,B 0,C 0,E1 0.1598,E2 90.072} C_DIS
LIN {X 4.6536,Y 0.9508,Z 23,A -2.5336,B 0,C 0,E1 0.1598,E2 90.0719} C_DIS
LIN {X 4.7445,Y 0.1918,Z 23,A -2.5625,B 0,C 0,E1 0.1598,E2 90.0719} C_DIS
LIN {X 4.7339,Y -0.3815,Z 23,A -2.5873,B 0,C 0,E1 0.1598,E2 90.0719} C_DIS
LIN {X 4.611,Y -1.1358,Z 23,A -2.6238,B 0,C 0,E1 0.1598,E2 90.0718} C_DIS
LIN {X 4.37,Y -1.8612,Z 23,A -2.6635,B 0,C 0,E1 0.1598,E2 90.0718} C_DIS
LIN {X 4.0151,Y -2.5382,Z 23,A -2.7053,B 0,C 0,E1 0.1598,E2 90.0718} C_DIS
LIN {X 3.5547,Y -3.1484,Z 23,A -2.7482,B 0,C 0,E1 0.1598,E2 90.0718} C_DIS
LIN {X 3.0054,Y -3.68,Z 23,A -2.791,B 0,C 0,E1 0.1598,E2 90.0718} C_DIS
LIN {X 2.3765,Y -4.1152,Z 23,A -2.8326,B 0,C 0,E1 0.1598,E2 90.0718} C_DIS
LIN {X 1.595,Y -4.4742,Z 23,A -2.8766,B 0,C 0,E1 0.1598,E2 90.0717} C_DIS
LIN {X 0.9506,Y -4.6542,Z 23,A -2.9079,B 0,C 0,E1 0.1598,E2 90.0717} C_DIS
LIN {X 0.1917,Y -4.7449,Z 23,A -2.9397,B 0,C 0,E1 0.1598,E2 90.0717} C_DIS
LIN {X 0.1917,Y -4.7449,Z 23,A -2.9397,B 0,C 0,E1 0.1598,E2 90.0717} C_DIS
Enddeposition()
LIN {X 0.0237,Y -5.6873,Z 23,A -2.9847,B 0,C 0,E1 0.1598,E2 90.0704} C_DIS
Startdeposition()
$VEL.CP = VEL_PRINT
LIN {X 0.9934,Y -5.5988,Z 23,A -2.9465,B 0,C 0,E1 0.1598,E2 90.0716} C_DIS
LIN {X 1.7488,Y -5.408,Z 23,A -2.9107,B 0,C 0,E1 0.1598,E2 90.0716} C_DIS
LIN {X 2.4714,Y -5.1172,Z 23,A -2.8719,B 0,C 0,E1 0.1598,E2 90.0717} C_DIS
LIN {X 3.1479,Y -4.7315,Z 23,A -2.8306,B 0,C 0,E1 0.1598,E2 90.0717} C_DIS
LIN {X 3.9131,Y -4.1297,Z 23,A -2.7768,B 0,C 0,E1 0.1598,E2 90.0717} C_DIS
LIN {X 4.6535,Y -3.2733,Z 23,A -2.7131,B 0,C 0,E1 0.1598,E2 90.0716} C_DIS
LIN {X 5.2202,Y -2.2627,Z 23,A -2.6491,B 0,C 0,E1 0.1598,E2 90.0716} C_DIS
LIN {X 5.5596,Y -1.186,Z 23,A -2.5907,B 0,C 0,E1 0.1598,E2 90.0714} C_DIS
LIN {X 5.6744,Y -0.3611,Z 23,A -2.5517,B 0,C 0,E1 0.1598,E2 90.0718} C_DIS
LIN {X 5.6358,Y 0.7893,Z 23,A -2.5039,B 0,C 0,E1 0.1598,E2 90.0715} C_DIS
LIN {X 5.2286,Y 2.2429,Z 23,A -2.4567,B 0,C 0,E1 0.1598,E2 90.0711} C_DIS
LIN {X 4.9559,Y 2.7857,Z 23,A -2.4446,B 0,C 0,E1 0.1598,E2 90.072} C_DIS
LIN {X 4.5088,Y 3.4602,Z 23,A -2.4324,B 0,C 0,E1 0.1598,E2 90.072} C_DIS
LIN {X 3.9715,Y 4.0651,Z 23,A -2.4266,B 0,C 0,E1 0.1598,E2 90.0721} C_DIS
LIN {X 3.3538,Y 4.5876,Z 23,A -2.4273,B 0,C 0,E1 0.1598,E2 90.0721} C_DIS
LIN {X 2.6683,Y 5.0172,Z 23,A -2.4344,B 0,C 0,E1 0.1598,E2 90.0722} C_DIS
LIN {X 1.929,Y 5.3456,Z 23,A -2.4478,B 0,C 0,E1 0.1598,E2 90.0722} C_DIS
LIN {X 1.1503,Y 5.5648,Z 23,A -2.4673,B 0,C 0,E1 0.1598,E2 90.0722} C_DIS
LIN {X 0.3486,Y 5.6717,Z 23,A -2.4923,B 0,C 0,E1 0.1598,E2 90.0722} C_DIS
LIN {X -0.4604,Y 5.6644,Z 23,A -2.5225,B 0,C 0,E1 0.1598,E2 90.0722} C_DIS
LIN {X -1.2601,Y 5.5418,Z 23,A -2.5572,B 0,C 0,E1 0.1598,E2 90.0722} C_DIS
LIN {X -2.0346,Y 5.3077,Z 23,A -2.5956,B 0,C 0,E1 0.1598,E2 90.0721} C_DIS
LIN {X -2.7678,Y 4.9652,Z 23,A -2.6371,B 0,C 0,E1 0.1598,E2 90.0721} C_DIS
LIN {X -3.4447,Y 4.5218,Z 23,A -2.6807,B 0,C 0,E1 0.1598,E2 90.0719} C_DIS
LIN {X -4.0514,Y 3.9863,Z 23,A -2.7256,B 0,C 0,E1 0.1598,E2 90.0718} C_DIS
LIN {X -4.5753,Y 3.3697,Z 23,A -2.7709,B 0,C 0,E1 0.1598,E2 90.0717} C_DIS
LIN {X -5.0085,Y 2.6865,Z 23,A -2.8157,B 0,C 0,E1 0.1598,E2 90.0716} C_DIS
LIN {X -5.3387,Y 1.9478,Z 23,A -2.859,B 0,C 0,E1 0.1598,E2 90.0715} C_DIS
LIN {X -5.561,Y 1.17,Z 23,A -2.8999,B 0,C 0,E1 0.1598,E2 90.0714} C_DIS
LIN {X -5.67,Y 0.3685,Z 23,A -2.9378,B 0,C 0,E1 0.1598,E2 90.0714} C_DIS
LIN {X -5.6663,Y -0.4404,Z 23,A -2.9718,B 0,C 0,E1 0.1598,E2 90.0713} C_DIS
LIN {X -5.5465,Y -1.2405,Z 23,A -3.0012,B 0,C 0,E1 0.1598,E2 90.0713} C_DIS
LIN {X -5.3145,Y -2.0157,Z 23,A -3.0254,B 0,C 0,E1 0.1598,E2 90.0713} C_DIS
LIN {X -4.9762,Y -2.7509,Z 23,A -3.0441,B 0,C 0,E1 0.1598,E2 90.0713} C_DIS
LIN {X -4.27,Y -3.7603,Z 23,A -3.0606,B 0,C 0,E1 0.1598,E2 90.071} C_DIS
LIN {X -3.4828,Y -4.495,Z 23,A -3.063,B 0,C 0,E1 0.1598,E2 90.0712} C_DIS
LIN {X -2.8659,Y -4.911,Z 23,A -3.0581,B 0,C 0,E1 0.1598,E2 90.0714} C_DIS
LIN {X -1.8145,Y -5.3937,Z 23,A -3.04,B 0,C 0,E1 0.1598,E2 90.0714} C_DIS
LIN {X -0.9063,Y -5.6103,Z 23,A -3.0159,B 0,C 0,E1 0.1598,E2 90.0715} C_DIS
LIN {X 0.0237,Y -5.6873,Z 23,A -2.9851,B 0,C 0,E1 0.1598,E2 90.0715} C_DIS
Enddeposition()
LIN {X 0.0237,Y -5.6873,Z 23,A -2.9851,B 0,C 0,E1 0.1598,E2 90.0715} C_DIS
Startdeposition()
$VEL.CP = VEL_PRINT
LIN {X -0.379,Y -6.6091,Z 23,A -3.0386,B 0,C 0,E1 0.1598,E2 90.071} C_DIS
LIN {X -1.1022,Y -6.531,Z 23,A -3.0623,B 0,C 0,E1 0.1598,E2 90.0715} C_DIS
LIN {X -2.1544,Y -6.2592,Z 23,A -3.0894,B 0,C 0,E1 0.1598,E2 90.0715} C_DIS
LIN {X -2.8626,Y -5.9691,Z 23,A -3.1031,B 0,C 0,E1 0.1598,E2 90.0714} C_DIS
LIN {X -3.5327,Y -5.5998,Z 23,A -3.112,B 0,C 0,E1 0.1598,E2 90.0714} C_DIS
LIN {X -4.1545,Y -5.1538,Z 23,A -3.1159,B 0,C 0,E1 0.1598,E2 90.0714} C_DIS
LIN {X -4.7218,Y -4.6401,Z 23,A -3.1149,B 0,C 0,E1 0.1598,E2 90.0713} C_DIS
LIN {X -5.2249,Y -4.0636,Z 23,A -3.109,B 0,C 0,E1 0.1598,E2 90.0713} C_DIS
LIN {X -5.658,Y -3.4328,Z 23,A -3.0982,B 0,C 0,E1 0.1598,E2 90.0713} C_DIS
LIN {X -6.0176,Y -2.7574,Z 23,A -3.0828,B 0,C 0,E1 0.1598,E2 90.0713} C_DIS
LIN {X -6.2947,Y -2.0442,Z 23,A -3.0629,B 0,C 0,E1 0.1598,E2 90.0713} C_DIS
LIN {X -6.4875,Y -1.3039,Z 23,A -3.0387,B 0,C 0,E1 0.1598,E2 90.0713} C_DIS
LIN {X -6.5958,Y -0.5466,Z 23,A -3.0107,B 0,C 0,E1 0.1598,E2 90.0713} C_DIS
LIN {X -6.6157,Y 0.2183,Z 23,A -2.9791,B 0,C 0,E1 0.1598,E2 90.0713} C_DIS
LIN {X -6.5471,Y 0.9805,Z 23,A -2.9444,B 0,C 0,E1 0.1598,E2 90.0713} C_DIS
LIN {X -6.3884,Y 1.729,Z 23,A -2.907,B 0,C 0,E1 0.1598,E2 90.0714} C_DIS
LIN {X -6.1468,Y 2.4551,Z 23,A -2.8675,B 0,C 0,E1 0.1598,E2 90.0714} C_DIS
LIN {X -5.8245,Y 3.149,Z 23,A -2.8264,B 0,C 0,E1 0.1598,E2 90.0716} C_DIS
LIN {X -5.4223,Y 3.8,Z 23,A -2.7841,B 0,C 0,E1 0.1598,E2 90.0716} C_DIS
LIN {X -4.9469,Y 4.3995,Z 23,A -2.7413,B 0,C 0,E1 0.1598,E2 90.0717} C_DIS
LIN {X -4.4062,Y 4.9409,Z 23,A -2.6986,B 0,C 0,E1 0.1598,E2 90.0718} C_DIS
LIN {X -3.8065,Y 5.4164,Z 23,A -2.6564,B 0,C 0,E1 0.1598,E2 90.0719} C_DIS
LIN {X -3.1559,Y 5.8187,Z 23,A -2.6155,B 0,C 0,E1 0.1598,E2 90.072} C_DIS
LIN {X -2.4631,Y 6.1438,Z 23,A -2.5762,B 0,C 0,E1 0.1598,E2 90.072} C_DIS
LIN {X -1.738,Y 6.3885,Z 23,A -2.5391,B 0,C 0,E1 0.1598,E2 90.0722} C_DIS
LIN {X -0.9887,Y 6.5441,Z 23,A -2.5049,B 0,C 0,E1 0.1598,E2 90.0722} C_DIS
LIN {X -0.2269,Y 6.6146,Z 23,A -2.4738,B 0,C 0,E1 0.1598,E2 90.0722} C_DIS
LIN {X 0.538,Y 6.5969,Z 23,A -2.4464,B 0,C 0,E1 0.1598,E2 90.0723} C_DIS
LIN {X 1.2954,Y 6.4898,Z 23,A -2.423,B 0,C 0,E1 0.1598,E2 90.0723} C_DIS
LIN {X 2.0358,Y 6.2974,Z 23,A -2.4038,B 0,C 0,E1 0.1598,E2 90.0723} C_DIS
LIN {X 2.7497,Y 6.0219,Z 23,A -2.3891,B 0,C 0,E1 0.1598,E2 90.0723} C_DIS
LIN {X 3.6978,Y 5.495,Z 23,A -2.3763,B 0,C 0,E1 0.1598,E2 90.0723} C_DIS
LIN {X 4.4473,Y 4.903,Z 23,A -2.3737,B 0,C 0,E1 0.1598,E2 90.0723} C_DIS
LIN {X 4.9828,Y 4.3579,Z 23,A -2.3771,B 0,C 0,E1 0.1598,E2 90.0723} C_DIS
LIN {X 5.4504,Y 3.7539,Z 23,A -2.3855,B 0,C 0,E1 0.1598,E2 90.0722} C_DIS
LIN {X 5.8469,Y 3.1009,Z 23,A -2.3986,B 0,C 0,E1 0.1598,E2 90.0722} C_DIS
LIN {X 6.1664,Y 2.4069,Z 23,A -2.4163,B 0,C 0,E1 0.1598,E2 90.0721} C_DIS
LIN {X 6.4025,Y 1.6803,Z 23,A -2.4384,B 0,C 0,E1 0.1598,E2 90.0721} C_DIS
LIN {X 6.5535,Y 0.9313,Z 23,A -2.4647,B 0,C 0,E1 0.1598,E2 90.072} C_DIS
LIN {X 6.617,Y 0.1701,Z 23,A -2.4947,B 0,C 0,E1 0.1598,E2 90.072} C_DIS
LIN {X 6.5911,Y -0.5934,Z 23,A -2.5281,B 0,C 0,E1 0.1598,E2 90.0719} C_DIS
LIN {X 6.4786,Y -1.3489,Z 23,A -2.5644,B 0,C 0,E1 0.1598,E2 90.0719} C_DIS
LIN {X 6.2821,Y -2.087,Z 23,A -2.603,B 0,C 0,E1 0.1598,E2 90.0719} C_DIS
LIN {X 6,Y -2.7972,Z 23,A -2.6436,B 0,C 0,E1 0.1598,E2 90.0718} C_DIS
LIN {X 5.6383,Y -3.4702,Z 23,A -2.6855,B 0,C 0,E1 0.1598,E2 90.0718} C_DIS
LIN {X 5.199,Y -4.0952,Z 23,A -2.7283,B 0,C 0,E1 0.1598,E2 90.0718} C_DIS
LIN {X 4.693,Y -4.6675,Z 23,A -2.7712,B 0,C 0,E1 0.1598,E2 90.0718} C_DIS
LIN {X 4.1249,Y -5.1782,Z 23,A -2.8138,B 0,C 0,E1 0.1598,E2 90.0717} C_DIS
LIN {X 3.5001,Y -5.6176,Z 23,A -2.8555,B 0,C 0,E1 0.1598,E2 90.0717} C_DIS
LIN {X 2.8291,Y -5.9828,Z 23,A -2.8956,B 0,C 0,E1 0.1598,E2 90.0717} C_DIS
LIN {X 2.1211,Y -6.2699,Z 23,A -2.9338,B 0,C 0,E1 0.1598,E2 90.0717} C_DIS
LIN {X 1.3843,Y -6.4713,Z 23,A -2.9694,B 0,C 0,E1 0.1598,E2 90.0717} C_DIS
LIN {X 0.6296,Y -6.5896,Z 23,A -3.0022,B 0,C 0,E1 0.1598,E2 90.0716} C_DIS
LIN {X 0.6296,Y -6.5896,Z 23,A -3.0022,B 0,C 0,E1 0.1598,E2 90.0716} C_DIS
Enddeposition()
LIN {X 0.0622,Y -7.5534,Z 23,A -3.0629,B 0,C 0,E1 0.1598,E2 90.0703} C_DIS
Startdeposition()
$VEL.CP = VEL_PRINT
LIN {X 0.8398,Y -7.51,Z 23,A -3.0336,B 0,C 0,E1 0.1598,E2 90.0715} C_DIS
LIN {X 1.9806,Y -7.289,Z 23,A -2.9825,B 0,C 0,E1 0.1598,E2 90.0715} C_DIS
LIN {X 2.7901,Y -7.0182,Z 23,A -2.9413,B 0,C 0,E1 0.1598,E2 90.0716} C_DIS
LIN {X 3.8757,Y -6.4878,Z 23,A -2.8788,B 0,C 0,E1 0.1598,E2 90.0716} C_DIS
LIN {X 4.7343,Y -5.885,Z 23,A -2.8216,B 0,C 0,E1 0.1598,E2 90.0716} C_DIS
LIN {X 5.3578,Y -5.3233,Z 23,A -2.7749,B 0,C 0,E1 0.1598,E2 90.0717} C_DIS
LIN {X 5.9146,Y -4.6955,Z 23,A -2.7277,B 0,C 0,E1 0.1598,E2 90.0717} C_DIS
LIN {X 6.3977,Y -4.0095,Z 23,A -2.6807,B 0,C 0,E1 0.1598,E2 90.0717} C_DIS
LIN {X 6.8048,Y -3.2758,Z 23,A -2.6345,B 0,C 0,E1 0.1598,E2 90.0717} C_DIS
LIN {X 7.1277,Y -2.5013,Z 23,A -2.5896,B 0,C 0,E1 0.1598,E2 90.0717} C_DIS
LIN {X 7.4318,Y -1.3789,Z 23,A -2.5303,B 0,C 0,E1 0.1598,E2 90.0716} C_DIS
LIN {X 7.5432,Y -0.4051,Z 23,A -2.485,B 0,C 0,E1 0.1598,E2 90.0718} C_DIS
LIN {X 7.5257,Y 0.7015,Z 23,A -2.4383,B 0,C 0,E1 0.1598,E2 90.0717} C_DIS
LIN {X 7.321,Y 1.8728,Z 23,A -2.3957,B 0,C 0,E1 0.1598,E2 90.0714} C_DIS
LIN {X 6.8821,Y 3.1254,Z 23,A -2.3587,B 0,C 0,E1 0.1598,E2 90.0715} C_DIS
LIN {X 6.2197,Y 4.2912,Z 23,A -2.3336,B 0,C 0,E1 0.1598,E2 90.0715} C_DIS
LIN {X 5.5145,Y 5.1664,Z 23,A -2.3229,B 0,C 0,E1 0.1598,E2 90.072} C_DIS
LIN {X 4.7485,Y 5.8738,Z 23,A -2.3213,B 0,C 0,E1 0.1598,E2 90.0722} C_DIS
LIN {X 4.0713,Y 6.3607,Z 23,A -2.3258,B 0,C 0,E1 0.1598,E2 90.0723} C_DIS
LIN {X 3.3452,Y 6.7711,Z 23,A -2.3352,B 0,C 0,E1 0.1598,E2 90.0723} C_DIS
LIN {X 2.3016,Y 7.1978,Z 23,A -2.3556,B 0,C 0,E1 0.1598,E2 90.0723} C_DIS
LIN {X 0.8351,Y 7.5106,Z 23,A -2.3966,B 0,C 0,E1 0.1598,E2 90.0723} C_DIS
LIN {X -0.4475,Y 7.5439,Z 23,A -2.4426,B 0,C 0,E1 0.1598,E2 90.0723} C_DIS
LIN {X -1.5604,Y 7.3939,Z 23,A -2.49,B 0,C 0,E1 0.1598,E2 90.0723} C_DIS
LIN {X -2.5321,Y 7.1202,Z 23,A -2.5374,B 0,C 0,E1 0.1598,E2 90.0722} C_DIS
LIN {X -3.4747,Y 6.712,Z 23,A -2.5894,B 0,C 0,E1 0.1598,E2 90.072} C_DIS
LIN {X -4.2917,Y 6.2194,Z 23,A -2.6403,B 0,C 0,E1 0.1598,E2 90.072} C_DIS
LIN {X -5.1336,Y 5.5457,Z 23,A -2.6996,B 0,C 0,E1 0.1598,E2 90.0717} C_DIS
LIN {X -5.7262,Y 4.9306,Z 23,A -2.7475,B 0,C 0,E1 0.1598,E2 90.0717} C_DIS
LIN {X -6.4268,Y 3.9744,Z 23,A -2.8134,B 0,C 0,E1 0.1598,E2 90.0714} C_DIS
LIN {X -6.9073,Y 3.0667,Z 23,A -2.8693,B 0,C 0,E1 0.1598,E2 90.0714} C_DIS
LIN {X -7.3293,Y 1.841,Z 23,A -2.9362,B 0,C 0,E1 0.1598,E2 90.0709} C_DIS
LIN {X -7.5282,Y 0.6161,Z 23,A -2.9951,B 0,C 0,E1 0.1598,E2 90.0707} C_DIS
LIN {X -7.5565,Y -0.1038,Z 23,A -3.0271,B 0,C 0,E1 0.1598,E2 90.0713} C_DIS
LIN {X -7.4421,Y -1.2878,Z 23,A -3.0723,B 0,C 0,E1 0.1598,E2 90.0707} C_DIS
LIN {X -7.1945,Y -2.3121,Z 23,A -3.1066,B 0,C 0,E1 0.1598,E2 90.0707} C_DIS
LIN {X -6.7686,Y -3.3509,Z 23,A -3.1348,B 0,C 0,E1 0.1598,E2 90.0708} C_DIS
LIN {X -6.3874,Y -4.0286,Z 23,A -3.1498,B 0,C 0,E1 0.1598,E2 90.0711} C_DIS
LIN {X -5.9393,Y -4.6639,Z 23,A -3.1602,B 0,C 0,E1 0.1598,E2 90.0711} C_DIS
LIN {X -5.4277,Y -5.2493,Z 23,A -3.1662,B 0,C 0,E1 0.1598,E2 90.0711} C_DIS
LIN {X -4.8614,Y -5.782,Z 23,A -3.168,B 0,C 0,E1 0.1598,E2 90.0711} C_DIS
LIN {X -4.2403,Y -6.2498,Z 23,A -3.165,B 0,C 0,E1 0.1598,E2 90.0712} C_DIS
LIN {X -3.2402,Y -6.8269,Z 23,A -3.1527,B 0,C 0,E1 0.1598,E2 90.0712} C_DIS
LIN {X -2.2467,Y -7.2099,Z 23,A -3.1326,B 0,C 0,E1 0.1598,E2 90.0713} C_DIS
LIN {X -1.4207,Y -7.4174,Z 23,A -3.1112,B 0,C 0,E1 0.1598,E2 90.0713} C_DIS
LIN {X -0.5763,Y -7.5294,Z 23,A -3.085,B 0,C 0,E1 0.1598,E2 90.0715} C_DIS
LIN {X -0.5763,Y -7.5294,Z 23,A -3.085,B 0,C 0,E1 0.1598,E2 90.0715} C_DIS
Enddeposition()
LIN {X 0.0908,Y -8.4894,Z 23,A -3.1003,B 0,C 0,E1 0.1598,E2 90.0703} C_DIS
Startdeposition()
$VEL.CP = VEL_PRINT
LIN {X -0.9129,Y -8.4373,Z 23,A -3.136,B 0,C 0,E1 0.1598,E2 90.0713} C_DIS
LIN {X -1.7073,Y -8.3122,Z 23,A -3.1599,B 0,C 0,E1 0.1598,E2 90.0713} C_DIS
LIN {X -2.4864,Y -8.1129,Z 23,A -3.18,B 0,C 0,E1 0.1598,E2 90.0713} C_DIS
LIN {X -3.2432,Y -7.8411,Z 23,A -3.1962,B 0,C 0,E1 0.1598,E2 90.0713} C_DIS
LIN {X -3.971,Y -7.4992,Z 23,A -3.2083,B 0,C 0,E1 0.1598,E2 90.0713} C_DIS
LIN {X -4.6633,Y -7.0901,Z 23,A -3.2164,B 0,C 0,E1 0.1598,E2 90.0712} C_DIS
LIN {X -5.3141,Y -6.6175,Z 23,A -3.2202,B 0,C 0,E1 0.1598,E2 90.0712} C_DIS
LIN {X -6.1536,Y -5.8492,Z 23,A -3.2183,B 0,C 0,E1 0.1598,E2 90.071} C_DIS
LIN {X -6.9004,Y -4.9417,Z 23,A -3.2072,B 0,C 0,E1 0.1598,E2 90.0708} C_DIS
LIN {X -7.3624,Y -4.2218,Z 23,A -3.194,B 0,C 0,E1 0.1598,E2 90.071} C_DIS
LIN {X -7.7498,Y -3.4592,Z 23,A -3.176,B 0,C 0,E1 0.1598,E2 90.071} C_DIS
LIN {X -8.0585,Y -2.6615,Z 23,A -3.1536,B 0,C 0,E1 0.1598,E2 90.071} C_DIS
LIN {X -8.2854,Y -1.8369,Z 23,A -3.1271,B 0,C 0,E1 0.1598,E2 90.071} C_DIS
LIN {X -8.4286,Y -0.9937,Z 23,A -3.0968,B 0,C 0,E1 0.1598,E2 90.071} C_DIS
LIN {X -8.4861,Y -0.1404,Z 23,A -3.0629,B 0,C 0,E1 0.1598,E2 90.0711} C_DIS
LIN {X -8.457,Y 0.7143,Z 23,A -3.0258,B 0,C 0,E1 0.1598,E2 90.0711} C_DIS
LIN {X -8.3412,Y 1.5617,Z 23,A -2.9858,B 0,C 0,E1 0.1598,E2 90.0712} C_DIS
LIN {X -8.1413,Y 2.3932,Z 23,A -2.9434,B 0,C 0,E1 0.1598,E2 90.0712} C_DIS
LIN {X -7.8592,Y 3.2006,Z 23,A -2.899,B 0,C 0,E1 0.1598,E2 90.0714} C_DIS
LIN {X -7.3985,Y 4.1654,Z 23,A -2.8412,B 0,C 0,E1 0.1598,E2 90.0712} C_DIS
LIN {X -6.8233,Y 5.0545,Z 23,A -2.7827,B 0,C 0,E1 0.1598,E2 90.0715} C_DIS
LIN {X -6.1331,Y 5.8679,Z 23,A -2.723,B 0,C 0,E1 0.1598,E2 90.0716} C_DIS
LIN {X -5.513,Y 6.4542,Z 23,A -2.6755,B 0,C 0,E1 0.1598,E2 90.0718} C_DIS
LIN {X -4.8372,Y 6.9754,Z 23,A -2.6287,B 0,C 0,E1 0.1598,E2 90.0719} C_DIS
LIN {X -4.1125,Y 7.426,Z 23,A -2.5829,B 0,C 0,E1 0.1598,E2 90.072} C_DIS
LIN {X -3.3461,Y 7.8016,Z 23,A -2.5388,B 0,C 0,E1 0.1598,E2 90.0721} C_DIS
LIN {X -2.5459,Y 8.0983,Z 23,A -2.4968,B 0,C 0,E1 0.1598,E2 90.0722} C_DIS
LIN {X -1.72,Y 8.3132,Z 23,A -2.4572,B 0,C 0,E1 0.1598,E2 90.0722} C_DIS
LIN {X -0.8764,Y 8.4431,Z 23,A -2.4206,B 0,C 0,E1 0.1598,E2 90.0723} C_DIS
LIN {X -0.0241,Y 8.4877,Z 23,A -2.3873,B 0,C 0,E1 0.1598,E2 90.0723} C_DIS
LIN {X 0.8284,Y 8.4475,Z 23,A -2.3575,B 0,C 0,E1 0.1598,E2 90.0724} C_DIS
LIN {X 1.8821,Y 8.2803,Z 23,A -2.3256,B 0,C 0,E1 0.1598,E2 90.0724} C_DIS
LIN {X 2.9243,Y 7.9656,Z 23,A -2.3004,B 0,C 0,E1 0.1598,E2 90.0724} C_DIS
LIN {X 3.6442,Y 7.663,Z 23,A -2.2866,B 0,C 0,E1 0.1598,E2 90.0724} C_DIS
LIN {X 4.3334,Y 7.296,Z 23,A -2.2767,B 0,C 0,E1 0.1598,E2 90.0724} C_DIS
LIN {X 4.9865,Y 6.8678,Z 23,A -2.2708,B 0,C 0,E1 0.1598,E2 90.0724} C_DIS
LIN {X 5.8495,Y 6.1533,Z 23,A -2.269,B 0,C 0,E1 0.1598,E2 90.0722} C_DIS
LIN {X 6.6361,Y 5.2918,Z 23,A -2.2764,B 0,C 0,E1 0.1598,E2 90.0721} C_DIS
LIN {X 7.1272,Y 4.6085,Z 23,A -2.2875,B 0,C 0,E1 0.1598,E2 90.0722} C_DIS
LIN {X 7.5486,Y 3.8802,Z 23,A -2.3029,B 0,C 0,E1 0.1598,E2 90.0722} C_DIS
LIN {X 7.8957,Y 3.1137,Z 23,A -2.3227,B 0,C 0,E1 0.1598,E2 90.0722} C_DIS
LIN {X 8.1653,Y 2.3166,Z 23,A -2.3466,B 0,C 0,E1 0.1598,E2 90.0721} C_DIS
LIN {X 8.3546,Y 1.4968,Z 23,A -2.3745,B 0,C 0,E1 0.1598,E2 90.0721} C_DIS
LIN {X 8.4623,Y 0.6623,Z 23,A -2.406,B 0,C 0,E1 0.1598,E2 90.072} C_DIS
LIN {X 8.4774,Y -0.481,Z 23,A -2.4538,B 0,C 0,E1 0.1598,E2 90.0716} C_DIS
LIN {X 8.3605,Y -1.4861,Z 23,A -2.501,B 0,C 0,E1 0.1598,E2 90.0716} C_DIS
LIN {X 8.1168,Y -2.486,Z 23,A -2.5526,B 0,C 0,E1 0.1598,E2 90.0716} C_DIS
LIN {X 7.8374,Y -3.2606,Z 23,A -2.596,B 0,C 0,E1 0.1598,E2 90.0718} C_DIS
LIN {X 7.4843,Y -4.0043,Z 23,A -2.6407,B 0,C 0,E1 0.1598,E2 90.0718} C_DIS
LIN {X 7.0605,Y -4.7102,Z 23,A -2.6863,B 0,C 0,E1 0.1598,E2 90.0718} C_DIS
LIN {X 6.4406,Y -5.5317,Z 23,A -2.7439,B 0,C 0,E1 0.1598,E2 90.0715} C_DIS
LIN {X 5.6298,Y -6.3566,Z 23,A -2.8088,B 0,C 0,E1 0.1598,E2 90.0715} C_DIS
LIN {X 4.793,Y -7.0067,Z 23,A -2.8673,B 0,C 0,E1 0.1598,E2 90.0715} C_DIS
LIN {X 4.0704,Y -7.45,Z 23,A -2.9128,B 0,C 0,E1 0.1598,E2 90.0715} C_DIS
LIN {X 3.307,Y -7.8187,Z 23,A -2.9565,B 0,C 0,E1 0.1598,E2 90.0715} C_DIS
LIN {X 2.5107,Y -8.1095,Z 23,A -2.9981,B 0,C 0,E1 0.1598,E2 90.0715} C_DIS
LIN {X 1.4814,Y -8.3612,Z 23,A -3.0465,B 0,C 0,E1 0.1598,E2 90.0715} C_DIS
LIN {X 0.3014,Y -8.482,Z 23,A -3.0949,B 0,C 0,E1 0.1598,E2 90.0715} C_DIS
LIN {X 0.3014,Y -8.482,Z 23,A -3.0949,B 0,C 0,E1 0.1598,E2 90.0715} C_DIS
Enddeposition()
LIN {X 0.0005,Y -4.7524,Z 24,A -2.9326,B 0,C 0,E1 0.1598,E2 90.0603} C_DIS
Startdeposition()
$VEL.CP = VEL_PRINT
LIN {X 0.0005,Y -4.7524,Z 24,A -2.9383,B 0,C 0,E1 0.1598,E2 90.0661} C_DIS
LIN {X 0.782,Y -4.6833,Z 24,A -2.9115,B 0,C 0,E1 0.1598,E2 90.071} C_DIS
LIN {X 1.5423,Y -4.4916,Z 24,A -2.8761,B 0,C 0,E1 0.1598,E2 90.0717} C_DIS
LIN {X 2.2606,Y -4.1762,Z 24,A -2.8364,B 0,C 0,E1 0.1598,E2 90.0717} C_DIS
LIN {X 2.7606,Y -3.8658,Z 24,A -2.8048,B 0,C 0,E1 0.1598,E2 90.0717} C_DIS
LIN {X 3.3602,Y -3.3595,Z 24,A -2.7612,B 0,C 0,E1 0.1598,E2 90.0717} C_DIS
LIN {X 3.8672,Y -2.7604,Z 24,A -2.7171,B 0,C 0,E1 0.1598,E2 90.0717} C_DIS
LIN {X 4.2673,Y -2.0856,Z 24,A -2.6736,B 0,C 0,E1 0.1598,E2 90.0717} C_DIS
LIN {X 4.5521,Y -1.3546,Z 24,A -2.632,B 0,C 0,E1 0.1598,E2 90.0717} C_DIS
LIN {X 4.7126,Y -0.5869,Z 24,A -2.5935,B 0,C 0,E1 0.1598,E2 90.0717} C_DIS
LIN {X 4.75,Y 0.0006,Z 24,A -2.5673,B 0,C 0,E1 0.1598,E2 90.072} C_DIS
LIN {X 4.7,Y 0.6853,Z 24,A -2.54,B 0,C 0,E1 0.1598,E2 90.072} C_DIS
LIN {X 4.5521,Y 1.3556,Z 24,A -2.5169,B 0,C 0,E1 0.1598,E2 90.072} C_DIS
LIN {X 4.2666,Y 2.0863,Z 24,A -2.4964,B 0,C 0,E1 0.1598,E2 90.072} C_DIS
LIN {X 3.8652,Y 2.7602,Z 24,A -2.4826,B 0,C 0,E1 0.1598,E2 90.072} C_DIS
LIN {X 3.3598,Y 3.3604,Z 24,A -2.4758,B 0,C 0,E1 0.1598,E2 90.072} C_DIS
LIN {X 2.7602,Y 3.8667,Z 24,A -2.4765,B 0,C 0,E1 0.1598,E2 90.0721} C_DIS
LIN {X 2.0857,Y 4.2676,Z 24,A -2.4844,B 0,C 0,E1 0.1598,E2 90.0721} C_DIS
LIN {X 1.3547,Y 4.5525,Z 24,A -2.4993,B 0,C 0,E1 0.1598,E2 90.0721} C_DIS
LIN {X 0.587,Y 4.7127,Z 24,A -2.5209,B 0,C 0,E1 0.1598,E2 90.0721} C_DIS
LIN {X -0.0006,Y 4.75,Z 24,A -2.541,B 0,C 0,E1 0.1598,E2 90.0721} C_DIS
LIN {X -0.782,Y 4.6833,Z 24,A -2.5726,B 0,C 0,E1 0.1598,E2 90.0721} C_DIS
LIN {X -1.5424,Y 4.4916,Z 24,A -2.6087,B 0,C 0,E1 0.1598,E2 90.0721} C_DIS
LIN {X -2.2606,Y 4.1763,Z 24,A -2.6485,B 0,C 0,E1 0.1598,E2 90.072} C_DIS
LIN {X -2.9171,Y 3.7472,Z 24,A -2.6908,B 0,C 0,E1 0.1598,E2 90.0719} C_DIS
LIN {X -3.4948,Y 3.2166,Z 24,A -2.7345,B 0,C 0,E1 0.1598,E2 90.0718} C_DIS
LIN {X -3.9758,Y 2.5969,Z 24,A -2.7783,B 0,C 0,E1 0.1598,E2 90.0717} C_DIS
LIN {X -4.3493,Y 1.9073,Z 24,A -2.8211,B 0,C 0,E1 0.1598,E2 90.0716} C_DIS
LIN {X -4.6038,Y 1.1653,Z 24,A -2.8618,B 0,C 0,E1 0.1598,E2 90.0715} C_DIS
LIN {X -4.7331,Y 0.3916,Z 24,A -2.8992,B 0,C 0,E1 0.1598,E2 90.0714} C_DIS
LIN {X -4.7478,Y -0.1968,Z 24,A -2.9247,B 0,C 0,E1 0.1598,E2 90.0714} C_DIS
LIN {X -4.6497,Y -0.9753,Z 24,A -2.9539,B 0,C 0,E1 0.1598,E2 90.0714} C_DIS
LIN {X -4.4248,Y -1.7271,Z 24,A -2.9774,B 0,C 0,E1 0.1598,E2 90.0714} C_DIS
LIN {X -4.0798,Y -2.4315,Z 24,A -2.9946,B 0,C 0,E1 0.1598,E2 90.0714} C_DIS
LIN {X -3.6233,Y -3.0694,Z 24,A -3.0048,B 0,C 0,E1 0.1598,E2 90.0714} C_DIS
LIN {X -3.2166,Y -3.4948,Z 24,A -3.008,B 0,C 0,E1 0.1598,E2 90.0714} C_DIS
LIN {X -2.5969,Y -3.9758,Z 24,A -3.0056,B 0,C 0,E1 0.1598,E2 90.0714} C_DIS
LIN {X -1.9073,Y -4.3493,Z 24,A -2.9961,B 0,C 0,E1 0.1598,E2 90.0714} C_DIS
LIN {X -1.1654,Y -4.6038,Z 24,A -2.9797,B 0,C 0,E1 0.1598,E2 90.0716} C_DIS
LIN {X -0.3917,Y -4.7331,Z 24,A -2.9568,B 0,C 0,E1 0.1598,E2 90.0716} C_DIS
LIN {X -0.3917,Y -4.7331,Z 24,A -2.9568,B 0,C 0,E1 0.1598,E2 90.0716} C_DIS
Enddeposition()
LIN {X 0.0361,Y -5.6893,Z 24,A -2.9806,B 0,C 0,E1 0.1598,E2 90.0704} C_DIS
Startdeposition()
$VEL.CP = VEL_PRINT
LIN {X -0.7882,Y -5.6359,Z 24,A -3.0097,B 0,C 0,E1 0.1598,E2 90.0715} C_DIS
LIN {X -2.1085,Y -5.2847,Z 24,A -3.0433,B 0,C 0,E1 0.1598,E2 90.0715} C_DIS
LIN {X -3.0302,Y -4.8153,Z 24,A -3.0572,B 0,C 0,E1 0.1598,E2 90.0714} C_DIS
LIN {X -3.8409,Y -4.1905,Z 24,A -3.0604,B 0,C 0,E1 0.1598,E2 90.0713} C_DIS
LIN {X -4.4029,Y -3.5952,Z 24,A -3.0559,B 0,C 0,E1 0.1598,E2 90.0713} C_DIS
LIN {X -4.8739,Y -2.9255,Z 24,A -3.0448,B 0,C 0,E1 0.1598,E2 90.0713} C_DIS
LIN {X -5.2429,Y -2.1947,Z 24,A -3.0274,B 0,C 0,E1 0.1598,E2 90.0713} C_DIS
LIN {X -5.5034,Y -1.4186,Z 24,A -3.0042,B 0,C 0,E1 0.1598,E2 90.0713} C_DIS
LIN {X -5.6505,Y -0.6134,Z 24,A -2.9755,B 0,C 0,E1 0.1598,E2 90.0713} C_DIS
LIN {X -5.6788,Y 0.2046,Z 24,A -2.942,B 0,C 0,E1 0.1598,E2 90.0713} C_DIS
LIN {X -5.5921,Y 1.0186,Z 24,A -2.9045,B 0,C 0,E1 0.1598,E2 90.0713} C_DIS
LIN {X -5.388,Y 1.8114,Z 24,A -2.8635,B 0,C 0,E1 0.1598,E2 90.0714} C_DIS
LIN {X -5.071,Y 2.5662,Z 24,A -2.82,B 0,C 0,E1 0.1598,E2 90.0715} C_DIS
LIN {X -4.6497,Y 3.268,Z 24,A -2.7749,B 0,C 0,E1 0.1598,E2 90.0716} C_DIS
LIN {X -3.9936,Y 4.0532,Z 24,A -2.7174,B 0,C 0,E1 0.1598,E2 90.0716} C_DIS
LIN {X -3.0814,Y 4.7775,Z 24,A -2.6533,B 0,C 0,E1 0.1598,E2 90.0718} C_DIS
LIN {X -2.3403,Y 5.1796,Z 24,A -2.6091,B 0,C 0,E1 0.1598,E2 90.072} C_DIS
LIN {X -1.5481,Y 5.4678,Z 24,A -2.5678,B 0,C 0,E1 0.1598,E2 90.0721} C_DIS
LIN {X -0.7223,Y 5.6366,Z 24,A -2.5302,B 0,C 0,E1 0.1598,E2 90.0721} C_DIS
LIN {X 0.1195,Y 5.6809,Z 24,A -2.4973,B 0,C 0,E1 0.1598,E2 90.0722} C_DIS
LIN {X 0.9584,Y 5.6002,Z 24,A -2.4698,B 0,C 0,E1 0.1598,E2 90.0722} C_DIS
LIN {X 1.7765,Y 5.3976,Z 24,A -2.4482,B 0,C 0,E1 0.1598,E2 90.0722} C_DIS
LIN {X 2.5551,Y 5.0748,Z 24,A -2.4331,B 0,C 0,E1 0.1598,E2 90.0722} C_DIS
LIN {X 3.2782,Y 4.6416,Z 24,A -2.4247,B 0,C 0,E1 0.1598,E2 90.0722} C_DIS
LIN {X 3.9283,Y 4.1051,Z 24,A -2.4235,B 0,C 0,E1 0.1598,E2 90.0722} C_DIS
LIN {X 4.4927,Y 3.4792,Z 24,A -2.4292,B 0,C 0,E1 0.1598,E2 90.0721} C_DIS
LIN {X 4.9599,Y 2.7774,Z 24,A -2.4417,B 0,C 0,E1 0.1598,E2 90.0721} C_DIS
LIN {X 5.2422,Y 2.211,Z 24,A -2.4555,B 0,C 0,E1 0.1598,E2 90.0721} C_DIS
LIN {X 5.5707,Y 1.1341,Z 24,A -2.4886,B 0,C 0,E1 0.1598,E2 90.0716} C_DIS
LIN {X 5.6712,Y 0.4011,Z 24,A -2.5164,B 0,C 0,E1 0.1598,E2 90.0719} C_DIS
LIN {X 5.6759,Y -0.3387,Z 24,A -2.5477,B 0,C 0,E1 0.1598,E2 90.0719} C_DIS
LIN {X 5.5839,Y -1.0728,Z 24,A -2.5823,B 0,C 0,E1 0.1598,E2 90.0719} C_DIS
LIN {X 5.3948,Y -1.7881,Z 24,A -2.6197,B 0,C 0,E1 0.1598,E2 90.0719} C_DIS
LIN {X 5.1195,Y -2.4747,Z 24,A -2.659,B 0,C 0,E1 0.1598,E2 90.0718} C_DIS
LIN {X 4.6534,Y -3.2735,Z 24,A -2.7099,B 0,C 0,E1 0.1598,E2 90.0716} C_DIS
LIN {X 3.8332,Y -4.2056,Z 24,A -2.7796,B 0,C 0,E1 0.1598,E2 90.0714} C_DIS
LIN {X 3.3456,Y -4.5963,Z 24,A -2.8144,B 0,C 0,E1 0.1598,E2 90.0717} C_DIS
LIN {X 2.6385,Y -5.0354,Z 24,A -2.8591,B 0,C 0,E1 0.1598,E2 90.0717} C_DIS
LIN {X 1.875,Y -5.367,Z 24,A -2.9012,B 0,C 0,E1 0.1598,E2 90.0717} C_DIS
LIN {X 1.0713,Y -5.5839,Z 24,A -2.94,B 0,C 0,E1 0.1598,E2 90.0717} C_DIS
LIN {X 0.0361,Y -5.6893,Z 24,A -2.9824,B 0,C 0,E1 0.1598,E2 90.0716} C_DIS
Enddeposition()
LIN {X 0.0361,Y -5.6893,Z 24,A -2.9824,B 0,C 0,E1 0.1598,E2 90.0716} C_DIS
Startdeposition()
$VEL.CP = VEL_PRINT
LIN {X 0.5998,Y -6.5907,Z 24,A -2.9996,B 0,C 0,E1 0.1598,E2 90.071} C_DIS
LIN {X 1.3517,Y -6.4783,Z 24,A -2.9678,B 0,C 0,E1 0.1598,E2 90.0716} C_DIS
LIN {X 2.0863,Y -6.2825,Z 24,A -2.9325,B 0,C 0,E1 0.1598,E2 90.0716} C_DIS
LIN {X 2.7925,Y -6.0007,Z 24,A -2.8946,B 0,C 0,E1 0.1598,E2 90.0716} C_DIS
LIN {X 3.4622,Y -5.6406,Z 24,A -2.8547,B 0,C 0,E1 0.1598,E2 90.0717} C_DIS
LIN {X 4.0878,Y -5.2084,Z 24,A -2.8134,B 0,C 0,E1 0.1598,E2 90.0717} C_DIS
LIN {X 4.6569,Y -4.7043,Z 24,A -2.771,B 0,C 0,E1 0.1598,E2 90.0717} C_DIS
LIN {X 5.1651,Y -4.1388,Z 24,A -2.7282,B 0,C 0,E1 0.1598,E2 90.0717} C_DIS
LIN {X 5.607,Y -3.52,Z 24,A -2.6857,B 0,C 0,E1 0.1598,E2 90.0717} C_DIS
LIN {X 5.9722,Y -2.8531,Z 24,A -2.6438,B 0,C 0,E1 0.1598,E2 90.0718} C_DIS
LIN {X 6.2596,Y -2.1492,Z 24,A -2.6033,B 0,C 0,E1 0.1598,E2 90.0718} C_DIS
LIN {X 6.4641,Y -1.4171,Z 24,A -2.5646,B 0,C 0,E1 0.1598,E2 90.0718} C_DIS
LIN {X 6.585,Y -0.6665,Z 24,A -2.5282,B 0,C 0,E1 0.1598,E2 90.0718} C_DIS
LIN {X 6.62,Y 0.0931,Z 24,A -2.4946,B 0,C 0,E1 0.1598,E2 90.0719} C_DIS
LIN {X 6.5646,Y 0.8515,Z 24,A -2.4644,B 0,C 0,E1 0.1598,E2 90.0719} C_DIS
LIN {X 6.4241,Y 1.5988,Z 24,A -2.4378,B 0,C 0,E1 0.1598,E2 90.072} C_DIS
LIN {X 6.1966,Y 2.3243,Z 24,A -2.4154,B 0,C 0,E1 0.1598,E2 90.072} C_DIS
LIN {X 5.8904,Y 3.0202,Z 24,A -2.3971,B 0,C 0,E1 0.1598,E2 90.072} C_DIS
LIN {X 5.5042,Y 3.6752,Z 24,A -2.3835,B 0,C 0,E1 0.1598,E2 90.0721} C_DIS
LIN {X 5.0461,Y 4.282,Z 24,A -2.3747,B 0,C 0,E1 0.1598,E2 90.0721} C_DIS
LIN {X 4.521,Y 4.8318,Z 24,A -2.3707,B 0,C 0,E1 0.1598,E2 90.0722} C_DIS
LIN {X 3.9386,Y 5.3205,Z 24,A -2.3715,B 0,C 0,E1 0.1598,E2 90.0722} C_DIS
LIN {X 3.3022,Y 5.7367,Z 24,A -2.3774,B 0,C 0,E1 0.1598,E2 90.0722} C_DIS
LIN {X 2.6229,Y 6.0787,Z 24,A -2.388,B 0,C 0,E1 0.1598,E2 90.0723} C_DIS
LIN {X 1.908,Y 6.3378,Z 24,A -2.4034,B 0,C 0,E1 0.1598,E2 90.0723} C_DIS
LIN {X 1.1688,Y 6.5158,Z 24,A -2.4232,B 0,C 0,E1 0.1598,E2 90.0723} C_DIS
LIN {X 0.4137,Y 6.6047,Z 24,A -2.4473,B 0,C 0,E1 0.1598,E2 90.0723} C_DIS
LIN {X -0.3464,Y 6.6091,Z 24,A -2.4752,B 0,C 0,E1 0.1598,E2 90.0723} C_DIS
LIN {X -1.1025,Y 6.5289,Z 24,A -2.5064,B 0,C 0,E1 0.1598,E2 90.0723} C_DIS
LIN {X -1.8432,Y 6.3573,Z 24,A -2.541,B 0,C 0,E1 0.1598,E2 90.0722} C_DIS
LIN {X -2.5595,Y 6.1027,Z 24,A -2.5782,B 0,C 0,E1 0.1598,E2 90.0722} C_DIS
LIN {X -3.2426,Y 5.769,Z 24,A -2.6174,B 0,C 0,E1 0.1598,E2 90.072} C_DIS
LIN {X -3.8834,Y 5.36,Z 24,A -2.6583,B 0,C 0,E1 0.1598,E2 90.072} C_DIS
LIN {X -4.4734,Y 4.8803,Z 24,A -2.7003,B 0,C 0,E1 0.1598,E2 90.0719} C_DIS
LIN {X -5.0042,Y 4.3359,Z 24,A -2.7428,B 0,C 0,E1 0.1598,E2 90.0718} C_DIS
LIN {X -5.4684,Y 3.7337,Z 24,A -2.7853,B 0,C 0,E1 0.1598,E2 90.0717} C_DIS
LIN {X -5.8594,Y 3.0815,Z 24,A -2.8272,B 0,C 0,E1 0.1598,E2 90.0716} C_DIS
LIN {X -6.1726,Y 2.3888,Z 24,A -2.8679,B 0,C 0,E1 0.1598,E2 90.0716} C_DIS
LIN {X -6.4048,Y 1.6649,Z 24,A -2.907,B 0,C 0,E1 0.1598,E2 90.0714} C_DIS
LIN {X -6.5552,Y 0.9197,Z 24,A -2.9439,B 0,C 0,E1 0.1598,E2 90.0714} C_DIS
LIN {X -6.6189,Y 0.1619,Z 24,A -2.9783,B 0,C 0,E1 0.1598,E2 90.0714} C_DIS
LIN {X -6.5924,Y -0.598,Z 24,A -3.0093,B 0,C 0,E1 0.1598,E2 90.0713} C_DIS
LIN {X -6.479,Y -1.3498,Z 24,A -3.0369,B 0,C 0,E1 0.1598,E2 90.0713} C_DIS
LIN {X -6.2823,Y -2.0842,Z 24,A -3.0607,B 0,C 0,E1 0.1598,E2 90.0713} C_DIS
LIN {X -6.0004,Y -2.7903,Z 24,A -3.0802,B 0,C 0,E1 0.1598,E2 90.0713} C_DIS
LIN {X -5.6407,Y -3.46,Z 24,A -3.0953,B 0,C 0,E1 0.1598,E2 90.0713} C_DIS
LIN {X -5.2077,Y -4.0849,Z 24,A -3.1059,B 0,C 0,E1 0.1598,E2 90.0713} C_DIS
LIN {X -4.7058,Y -4.6561,Z 24,A -3.1116,B 0,C 0,E1 0.1598,E2 90.0713} C_DIS
LIN {X -4.14,Y -5.1641,Z 24,A -3.1124,B 0,C 0,E1 0.1598,E2 90.0713} C_DIS
LIN {X -3.5202,Y -5.6046,Z 24,A -3.1083,B 0,C 0,E1 0.1598,E2 90.0713} C_DIS
LIN {X -2.8542,Y -5.9714,Z 24,A -3.0995,B 0,C 0,E1 0.1598,E2 90.0713} C_DIS
Enddeposition()
END
